# B&R Automation Studio project AAU12Segmenter (part 8)

#### mxA_Start.st
```iecst
ACTION mxA_Start:

	/////////////////////////////////////////////////////
	// Logic to call the KRC_Initialize				   //
	// KRC_Initialize gives back the Status of the	   //
	// like, online, Initialized,.......			   //
	/////////////////////////////////////////////////////

	KRC_Initialize_0.AxisGroupIdx 			:= 1;
	KRC_Initialize_0.KRC_AxisGroupRefArr 	:= ADR(AxisRef);
	HMI_R1_Init_Done 						:=	KRC_Initialize_0.Done;
	HMI_R1_Init_Error 						:=	KRC_Initialize_0.Error;
	HMI_R1_Init_Error_ID 					:=	KRC_Initialize_0.ErrorID;

	KRC_Initialize_0();

	KRC_Initialize_1.AxisGroupIdx 			:= 2;
	KRC_Initialize_1.KRC_AxisGroupRefArr 	:= ADR(AxisRef);
	HMI_R2_Init_Done 						:=	KRC_Initialize_1.Done;
	HMI_R2_Init_Error 						:=	KRC_Initialize_1.Error;
	HMI_R2_Init_Error_ID 					:=	KRC_Initialize_1.ErrorID;

	KRC_Initialize_1();

	/////////////////////////////////////////////////////
	// Logic to call the KRC_Error     			       //
	// KRC_Error gives back the Status of the Robot    //
	// like, online, Initialized,.......			   //
	/////////////////////////////////////////////////////

	KRC_Error_0.AxisGroupIdx 				:= 1;
	KRC_Error_0.MessageReset 				:= HMI_R1_MessageReset;
	KRC_Error_0.KRC_AxisGroupRefArr			:= ADR(AxisRef);
	HMI_R1_Error_General					:= KRC_Error_0.Error;
	HMI_R1_Error_General_ID					:= KRC_Error_0.ErrorID;
	HMI_R1_Error_Activ						:= KRC_Error_0.KrcErrorActive;
	HMI_R1_Error_DrivesNotReady				:= KRC_Error_0.DrivesNotReady;

	KRC_Error_0();

	KRC_Error_1.AxisGroupIdx 				:= 2;
	KRC_Error_1.MessageReset 				:= HMI_R2_MessageReset;
	KRC_Error_1.KRC_AxisGroupRefArr			:= ADR(AxisRef);
	HMI_R2_Error_General					:= KRC_Error_1.Error;
	HMI_R2_Error_General_ID					:= KRC_Error_1.ErrorID;
	HMI_R2_Error_Activ						:= KRC_Error_1.KrcErrorActive;
	HMI_R2_Error_DrivesNotReady				:= KRC_Error_1.DrivesNotReady;

	KRC_Error_1();

	//////////////////////////////////////////////////////
	// KRC_AutomaticExternal allows to control the 		//
	// Robot with the PLC								//
	//////////////////////////////////////////////////////

	KRC_AutomaticExternal_0.AxisGroupIdx 		:= 1;
	KRC_AutomaticExternal_0.MOVE_ENABLE 		:= TRUE;
	KRC_AutomaticExternal_0.DRIVES_OFF 			:= TRUE;
	KRC_AutomaticExternal_0.KRC_AxisGroupRefArr	:= ADR(AxisRef);
	KRC_AutomaticExternal_0.EXT_START 			:= HMI_R1_EXT_START;
	KRC_AutomaticExternal_0.ENABLE_T1 			:= TRUE;
	KRC_AutomaticExternal_0.ENABLE_EXT 			:= TRUE;

	KRC_AutomaticExternal_0();

	KRC_AutomaticExternal_1.AxisGroupIdx 		:= 2;
	KRC_AutomaticExternal_1.MOVE_ENABLE 		:= TRUE;
	KRC_AutomaticExternal_1.DRIVES_OFF 			:= TRUE;
	KRC_AutomaticExternal_1.KRC_AxisGroupRefArr := ADR(AxisRef);
	KRC_AutomaticExternal_1.EXT_START			:= HMI_R2_EXT_START;
	KRC_AutomaticExternal_1.ENABLE_T1 			:= TRUE;
	KRC_AutomaticExternal_1.ENABLE_EXT 			:= TRUE;

	KRC_AutomaticExternal_1();

	//////////////////////////////////////////////////////
	//Function Block for StartUp of Robot				//
	//////////////////////////////////////////////////////

	KRC_AutoStart_0.AxisGroupIdx 				:= 1;
	KRC_AutoStart_0.KRC_AxisGroupRefArr 		:= ADR(AxisRef);
	KRC_AutoStart_0.ExecuteReset 				:= HMI_R1_AutoStart ;

	KRC_AutoStart_0();

	KRC_AutoStart_1.AxisGroupIdx 				:= 2;
	KRC_AutoStart_1.KRC_AxisGroupRefArr 		:= ADR(AxisRef);
	KRC_AutoStart_1.ExecuteReset 				:= HMI_R2_AutoStart ;

	KRC_AutoStart_1();

	//////////////////////////////////////////////////////
	// KRC_SetOverride used to set the Override 		//
	// for the Robot Velocity							//
	//////////////////////////////////////////////////////

	KRC_SetOverride_0.AxisGroupIdx 				:= 1;
	KRC_SetOverride_0.KRC_AxisGroupRefArr 		:= ADR(AxisRef);
	KRC_SetOverride_0.Override 					:= HMI_R1_Override;

	KRC_SetOverride_0();

	KRC_SetOverride_1.AxisGroupIdx 				:= 2;
	KRC_SetOverride_1.KRC_AxisGroupRefArr 		:= ADR(AxisRef);
	KRC_SetOverride_1.Override 					:=HMI_R2_Override;

	KRC_SetOverride_1();

	//////////////////////////////////////////////////////
	//KRC_Diag gives back some information about the 	//
	//axis and robot									//
	//////////////////////////////////////////////////////

	KRC_Diag_0.AxisGroupIdx 					:= 1;
	KRC_Diag_0.KRC_AxisGroupRefArr 				:= ADR(AxisRef);
	KRC_Diag_0.ShowTrace 						:= FALSE;

	KRC_Diag_0();

	KRC_Diag_1.AxisGroupIdx 					:= 2;
	KRC_Diag_1.KRC_AxisGroupRefArr 				:= ADR(AxisRef);
	KRC_Diag_1.ShowTrace 						:= FALSE;

	KRC_Diag_1();

	//////////////////////////////////////////////////////
	//Checking status of KRC and PLC for creating the   //
	//signals for the HMI 								//
	//										 			//
	//////////////////////////////////////////////////////

	CASE HMI_AxisGroup OF

	//////////////////////////////////////////////////////
	//ROBOT 1											//
	//////////////////////////////////////////////////////

		1:
			IF KRC_Diag_0.ProconosCyc_Act = -1 OR KRC_Error_0.NoHeartbeatPCOS THEN
				Status_P := FALSE;
			ELSE
				Status_P := TRUE;
			END_IF

			IF KRC_Diag_0.SubmitCyc_Act = -1 OR KRC_Error_0.NoHeartbeatKRC THEN
				Status_S := FALSE;
			ELSE
				Status_S := TRUE;
			END_IF

			IF KRC_AutomaticExternal_0.EXT THEN
				Status_EXT := 1;
			ELSE
				Status_EXT := 0;
			END_IF

			IF NOT KRC_Error_0.DrivesNotReady AND KRC_AutomaticExternal_0.RC_RDY1 THEN
				Status_I := 1;
			ELSE
				Status_I := 0;
			END_IF

			IF KRC_AutoStart_0.DispActive THEN
				Status_R	:= 1;
			ELSE
				Status_R	:= 0;
			END_IF

	//////////////////////////////////////////////////////
	//ROBOT 2											//
	//////////////////////////////////////////////////////

		2:
			IF KRC_Diag_1.ProconosCyc_Act = -1 OR KRC_Error_1.NoHeartbeatPCOS THEN
				Status_P := FALSE;
			ELSE
				Status_P := TRUE;
			END_IF

			IF KRC_Diag_1.SubmitCyc_Act = -1 OR KRC_Error_1.NoHeartbeatKRC THEN
				Status_S := FALSE;
			ELSE
				Status_S := TRUE;
			END_IF

			IF KRC_AutomaticExternal_1.EXT THEN
				Status_EXT := 1;
			ELSE
				Status_EXT := 0;
			END_IF

			IF NOT KRC_Error_1.DrivesNotReady AND KRC_AutomaticExternal_1.RC_RDY1 THEN
				Status_I := 1;
			ELSE
				Status_I := 0;
			END_IF

			IF KRC_AutoStart_1.DispActive THEN
				Status_R	:= 1;
			ELSE
				Status_R	:= 0;
			END_IF

	//////////////////////////////////////////////////////
	//ROBOT 3,4,5										//
	//////////////////////////////////////////////////////

		3,4,5:

			Status_P := FALSE;
			Status_S := FALSE;
			Status_I := 0;
			Status_R := 0;
			Status_EXT := 0;

	END_CASE;

END_ACTION
```

#### mxA_LinearMovement.st
```iecst
ACTION mxA_LinearMovement:

	CASE pState OF

		0:
			// Waiting for robot 1 to be ready to move
			IF 	Status_P > 0 AND Status_S > 0 AND Status_I > 0 AND Status_R > 0 AND Status_EXT > 0 THEN
				pState := 20;
			END_IF

		10:
			toolCover.X := 0;
			toolCover.Y := 0;
			toolCover.Z := 100;
			toolCover.A := 0;
			toolCover.B := 0;
			toolCover.C := 0;

			KRC_WriteToolData_0.AxisGroupIdx 		:= HMI_AxisGroup;
			KRC_WriteToolData_0.KRC_AxisGroupRefArr := ADR(AxisRef);
			KRC_WriteToolData_0.ToolNo 				:= 1;
			KRC_WriteToolData_0.ToolData 			:= toolCover;
			KRC_WriteToolData_0.BufferMode 			:= 2;
			KRC_WriteToolData_0.ExecuteCmd			:= TRUE;

			IF KRC_WriteToolData_0.Done THEN
				KRC_WriteToolData_0.ExecuteCmd		:= FALSE;
				pState := 20;
			END_IF

		20:

			//Set frames as coordsys
			mxa_ValuesToCOORDSYS_0.Tool 	:= 1; // Change to 1 when it works
			mxa_ValuesToCOORDSYS_0.Base 	:= 1;
			mxa_ValuesToCOORDSYS_0.IPO_Mode := 0;

			pState := 30;

		30:

			coordSys := mxa_ValuesToCOORDSYS_0.COORDSYS;

			KRC_MoveLinearAbsolute_0.AxisGroupIdx 			:= HMI_AxisGroup;
			KRC_MoveLinearAbsolute_0.KRC_AxisGroupRefArr	:= ADR(AxisRef);
			KRC_MoveLinearAbsolute_0.Velocity				:= 10;
			KRC_MoveLinearAbsolute_0.Acceleration  			:= 20;
			KRC_MoveLinearAbsolute_0.CoordinateSystem		:= coordSys;
			KRC_MoveLinearAbsolute_0.OriType 				:= 0;
			KRC_MoveLinearAbsolute_0.BufferMode				:= 2;

			pState := 40;

		40:
			endPOS.X := 302;
			endPOS.Y := -2;
			endPOS.Z := 527;
			endPOS.A := -178;
			endPOS.B := 26;
			endPOS.C := -178;
			endPOS.Status := 2; //010
			endPOS.Turn := 2; //000010

			KRC_MoveLinearAbsolute_0.Position			:= endPOS;

			KRC_MoveLinearAbsolute_0.ExecuteCmd 		:= TRUE;
			IF KRC_MoveLinearAbsolute_0.Done THEN
				KRC_MoveLinearAbsolute_0.ExecuteCmd 	:= FALSE;
				pState 									:= 50;
			END_IF

		50:
			endPOS.X := 430;
			endPOS.Y := -2;
			endPOS.Z := 527;
			endPOS.A := -178;
			endPOS.B := 26;
			endPOS.C := -178;
			endPOS.Status := 2; //010
			endPOS.Turn := 2; //000010

			KRC_MoveLinearAbsolute_0.Position			:= endPOS;

			KRC_MoveLinearAbsolute_0.ExecuteCmd 		:= TRUE;
			IF KRC_MoveLinearAbsolute_0.Done THEN
				KRC_MoveLinearAbsolute_0.ExecuteCmd 	:= FALSE;
				pState 									:= 40;
			END_IF

	END_CASE

	KRC_WriteToolData_0();
	mxa_ValuesToCOORDSYS_0();
	KRC_MoveLinearAbsolute_0();

END_ACTION
```

### Variables.var - Global variables
```iecst
(*********************************************************************************
 * Copyright: Bernecker + Rainer
 * Author:    reschl
 * Created:   July 02, 2015/4:23 PM
 *********************************************************************************
 * Global variables of project
 *********************************************************************************)
(*KRC <----> PLC communication*)
VAR
	KRC_Input : ARRAY[0..5,0..253] OF BYTE;
	KRC_Output : ARRAY[0..5,0..253] OF BYTE;
	InputVariables : ARRAY[0..5,0..253] OF USINT;
	OutputVariables : ARRAY[0..5,0..253] OF USINT;
	KUKAs : ARRAY[0..5] OF KUKA;
	KRC4_Input_1 : ARRAY[0..254] OF BYTE; (*Variable with the BYTE information from KRC*)
	KRC4_Input : ARRAY[0..254] OF BYTE; (*Variable with the BYTE information from KRC*)
	KRC4_Output_1 : ARRAY[0..254] OF BYTE; (*Variable with the BYTE information to KRC*)
	KRC4_Output : ARRAY[0..254] OF BYTE; (*Variable with the BYTE infromation to KRC*)
	InputVariablePL_1 : ARRAY[0..255] OF USINT;
	InputVariablePL : ARRAY[0..255] OF USINT;
	OutputVariablePL_1 : ARRAY[0..255] OF USINT;
	OutputVariablePL : ARRAY[0..255] OF USINT;
END_VAR
(*PositonArray, Coordsys etc*)
VAR RETAIN
	TeachPosition : POSITION_ARRAY; (*TeachingPositions -> retain to be save when restarting*)
END_VAR
VAR
	JogPosAxis : E6AXIS := (A2:=-90,A3:=90);
	JoggingCoordSys : COORDSYS; (*Variable for the CoordSystem when Jogging*)
	Coordsys_1 : COORDSYS;
END_VAR
VAR RETAIN
	gParameter : USINT;
END_VAR
(*HMI Variablen*)
VAR
	gCurrentPage : INT; (*Shows current page index of the Visualization*)
	HMI_Base_act : INT;
	HMI_Tool_act : INT;
	HMI_ExeAbort : BOOL;
	HMI_ExeMoveDirect : BOOL;
	HMI_AxisGroup : INT;
	HMI_R2_MessageReset : BOOL;
	HMI_R2_Override : INT;
	HMI_R2_AutoStart : BOOL;
	HMI_R2_EXT_START : BOOL;
	HMI_R2_Error_DrivesNotReady : BOOL;
	HMI_R2_Error_Activ : BOOL;
	HMI_R2_Error_General_ID : DINT;
	HMI_R2_Error_General : BOOL;
	HMI_R2_Init_Error_ID : DINT;
	HMI_R2_Init_Error : BOOL;
	HMI_R2_Init_Done : BOOL;
	HMI_R1_MessageReset : BOOL;
	HMI_R1_Override : INT;
	HMI_R1_AutoStart : BOOL;
	HMI_R1_EXT_START : BOOL;
	HMI_R1_Error_DrivesNotReady : BOOL;
	HMI_R1_Error_Activ : BOOL;
	HMI_R1_Error_General_ID : DINT;
	HMI_R1_Error_General : BOOL;
	HMI_R1_Init_Error_ID : DINT;
	HMI_R1_Init_Error : BOOL;
	HMI_R1_Init_Done : BOOL;
	HMI_A6 : REAL;
	HMI_A5 : REAL;
	HMI_A4 : REAL;
	HMI_A3 : REAL;
	HMI_A2 : REAL;
	HMI_A1 : REAL;
	HMI_C : REAL;
	HMI_B : REAL;
	HMI_A : REAL;
	HMI_Z : REAL;
	HMI_Y : REAL;
	HMI_X : REAL;
	HMI_A6_C_M : BOOL;
	HMI_A6_C_P : BOOL;
	HMI_A5_B_M : BOOL;
	HMI_A5_B_P : BOOL;
	HMI_A4_A_M : BOOL;
	HMI_A4_A_P : BOOL;
	HMI_A3_Z_M : BOOL;
	HMI_A3_Z_P : BOOL;
	HMI_A2_Y_M : BOOL;
	HMI_A2_Y_P : BOOL;
	HMI_A1_X_M : BOOL;
	HMI_A1_X_P : BOOL;
	HMI_Increment : INT;
	HMI_MoveType : INT;
END_VAR
```

### Types.typ - Global data types
```iecst
TYPE
	KUKA : 	STRUCT
		cm : brdkCM; (*Change type after integration into Smart Lab project*)
		init : init_function;
		motion : motion_function;
		read : read_function;
		operationType : operation_type;
		gripperType : gripper_type;
		TON_Timer : TON;
		operationDone : BOOL := FALSE; (*Maybe don't need. Depends how we send finish flag to ACOPOS*)
		status : status;
	END_STRUCT;
	init_function : 	STRUCT
		KRC_ReadAxisGroup : KRC_ReadAxisGroup;
		KRC_Initialize : KRC_Initialize;
		KRC_Error : KRC_Error;
		KRC_AutomaticExternal : KRC_AutomaticExternal;
		KRC_AutoStart : KRC_AutoStart;
		KRC_SetOverride : KRC_SetOverride;
		KRC_Diag : KRC_Diag;
		KRC_WriteAxisGroup : KRC_WriteAxisGroup;
	END_STRUCT;
	motion_function : 	STRUCT
		KRC_MoveDirectAbsolute : KRC_MoveDirectAbsolute;
		KRC_MoveDirectRelative : KRC_MoveDirectRelative;
		KRC_MoveLinearAbsolute : KRC_MoveLinearAbsolute;
		KRC_MoveLinearRelative : KRC_MoveLinearRelative;
	END_STRUCT;
	read_function : 	STRUCT
		KRC_ReadActualPosition : KRC_ReadActualPosition;
		KRC_ReadActualAxisPosition : KRC_ReadActualAxisPosition;
	END_STRUCT;
	operation_type :
		(
		ASSEMBLY := 0,
		PROCESS := 1
		);
	gripper_type :
		(
		COVER_GRIPPER := 0,
		PCB_GRIPPER := 1,
		FUSE_GRIPPER := 2
		);
	status : 	STRUCT
		S_ : BOOL;
		I_ : BOOL;
		R_ : BOOL;
		EXT_ : BOOL;
		P_ : BOOL;
	END_STRUCT;
END_TYPE
```

### Program Logical/Modules/KUKA/KUKA (IEC)

#### Types.typ - Local data types
```iecst
TYPE
	KUKA : 	STRUCT
		axisGroupIdx : USINT;
		startState : USINT;
		cm : brdkCM;
		start : start_function;
		motion : motion_function;
		convert : convert_function;
		read : read_function;
		write : write_function;
		status : status;
		operationType : operation_type;
		eeType : end_effector_type;
		gripperAction : GripperAction;
		tempPosition : E6POS;
		TON : TON;
	END_STRUCT;
	start_function : 	STRUCT
		KRC_Initialize : KRC_Initialize;
		KRC_Error : KRC_Error;
		KRC_AutomaticExternal : KRC_AutomaticExternal;
		KRC_AutoStart : KRC_AutoStart;
		KRC_SetOverride : KRC_SetOverride;
		KRC_Diag : KRC_Diag;
		KRC_Abort : KRC_Abort;
	END_STRUCT;
	motion_function : 	STRUCT
		KRC_MoveDirectAbsolute : KRC_MoveDirectAbsolute; (*PTP absolute motion*)
		KRC_MoveDirectRelative : KRC_MoveDirectRelative; (*PTP relative motion*)
		KRC_MoveLinearAbsolute : KRC_MoveLinearAbsolute; (*LIN absolute motion*)
		KRC_MoveLinearRelative : KRC_MoveLinearRelative; (*LIN relative motion*)
		KRC_MoveAxisAbsolute : KRC_MoveAxisAbsolute; (*JOINT absolute motion*)
	END_STRUCT;
	convert_function : 	STRUCT
		ValuesToCOORDSYS : mxa_ValuesToCOORDSYS;
		ValuesToPosition : ValuesToPosition;
		ValuesToMagazineFrame : ValuesToMagazineFrame;
	END_STRUCT;
	read_function : 	STRUCT
		KRC_ReadAxisGroup : KRC_ReadAxisGroup;
		KRC_ReadActualPosition : KRC_ReadActualPosition;
		KRC_ReadActualAxisPosition : KRC_ReadActualAxisPosition;
	END_STRUCT;
	write_function : 	STRUCT
		KRC_WriteAxisGroup : KRC_WriteAxisGroup;
		KRC_WriteToolData : KRC_WriteToolData;
		KRC_WriteBaseData : KRC_WriteBaseData;
	END_STRUCT;
	status : 	STRUCT
		S_ : BOOL;
		I_ : BOOL;
		R_ : BOOL;
		EXT_ : BOOL;
		P_ : BOOL;
	END_STRUCT;
	operation_type :
		(
		ASSEMBLY := 0,
		PROCESS := 1
		);
	end_effector_type :
		(
		COVER_EE := 1,
		PCB_EE := 2,
		FUSE_EE := 3,
		DRILL_EE := 4
		);
	gripper_action_type :
		(
		OPEN := 0,
		CLOSE := 1
		);
	robot_position_type :
		(
		DEFAULT := 0,
		APPROACH_MAGAZINE := 1,
		APPROACH_WORKSTATION := 2
		);
END_TYPE
```

#### Variables.var - Local variables
```iecst
VAR
	KUKAs : ARRAY[0..5] OF KUKA;
END_VAR
(*AxisStructure*)
VAR
	AxisRef : AXIS_GROUP_REF_ARR; (*Axis Reference of the Robot*)
END_VAR
(*Instance of FB*)
VAR
	mxa_ValuesToCOORDSYS_0 : mxa_ValuesToCOORDSYS;
	EETypeToFrame_0 : EETypeToFrame;
END_VAR
(*Variables for UDP-communication*)
VAR
	i : USINT; (*IndexVariable for ErrorMessages*)
	InputUDPString : STRING[255]; (*Variable with Message from KRC*)
	counterMsg : INT;
	WorkAroundCounter : INT;
	step_UDPConnect : INT; (*State-Variable for Errorhandling*)
	TextArray : ARRAY[0..15] OF STRING[255]; (*TextArray contains Messages from KRC*)
	UdpOpen_0 : UdpOpen; (*FunctionBlock to Open Port*)
	UdpOpen_1 : UdpOpen; (*FunctionBlock to Open Port*)
	UdpRecv_0 : UdpRecv; (*FunctionBlock to Receive Message*)
	UdpSend_0 : UdpSend; (*FunctionBlock to Send Message*)
	MsgToKrc : STRING[17]; (*Contains the Message which is send to KRC for getting all Messages*)
	ReloadMsg : BOOL; (*Variable triggers the Sequence to get Messages*)
END_VAR
VAR CONSTANT
	STATE_DISPLAY : INT := 5; (*STATE to display the Message*)
	STATE_RECEIVE : INT := 3; (*STATE to receive a new Message*)
	STATE_OPEN : INT := 0; (*STATE for opening the Ports*)
	STATE_SEND : INT := 2; (*STATE for sending a request to KRC*)
	STATE_WAIT : INT := 1; (*STATE for Waiting to trigger a new Request*)
END_VAR
VAR
	TON_0 : TON;
END_VAR
(*Misc*)
VAR
	acoposBase : FRAME;
	bottomCoverMagazineBase : FRAME;
	pcbMagazineBase : FRAME;
	fuseMagazineBase : FRAME;
	topCoverMagazineBase : FRAME;
	unloadingBase : FRAME;
	coordSys : COORDSYS;
	endPOS : E6POS;
	position1 : E6AXIS;
	position2 : E6AXIS;
END_VAR
(*For robot operations*)
VAR
	gripperWaitTime : INT;
END_VAR
VAR CONSTANT
	relativeDistance : REAL := 80.0;
	relativeDrillDistance : REAL := 10.0;
END_VAR
VAR
	drillYOffset : REAL := 27*2;
	drillXOffset : REAL := 53*2;
	numDoneHoles : USINT := 0;
	fusePickOffset : REAL := 13; (*Distance between fuses*)
	k : INT;
END_VAR
VAR CONSTANT
	unloadSizeX : INT := 2;
	unloadSizeY : INT := 2;
	unloadSizeZ : INT := 4;
END_VAR
VAR
	stackCounter : ARRAY[0..1,0..1] OF INT := [4(0)];
	idAtStack : ARRAY[0..1,0..1] OF INT := [4(-1)];
	xIdx : INT;
	yIdx : INT;
	xIdxTemp : INT := -1;
	yIdxTemp : INT := -1;
	orderCounter : ARRAY[0..1,0..1] OF INT := [4(0)];
END_VAR
(*References*)
VAR
	pKuka : REFERENCE TO KUKA;
	cm : REFERENCE TO brdkCM;
END_VAR
(*Variable mapping*)
VAR
	orderAmount : SINT;
	orderSpec : ARRAY[0..5] OF SINT;
	robotExecute : ARRAY[0..5] OF BOOL;
	robotDone : ARRAY[0..5] OF BOOL;
	robotBusy : ARRAY[0..5] OF BOOL;
END_VAR
```

#### Main.st - Cyclic code
```iecst
PROGRAM _INIT

	FOR i := 0 TO 5 DO
		KUKAs[i].axisGroupIdx := i + 1;
		KUKAs[i].gripperAction.whitePin := ADR(gripperWhitePins[i]);
		KUKAs[i].gripperAction.blackPin := ADR(gripperBlackPins[i]);
		KUKAs[i].gripperAction.action := OPEN;
		KUKAs[i].gripperAction();
		KUKAs[i].cm.state := 0;
		KUKAs[i].startState := 0;
	END_FOR

	// Setting end-effector type
	KUKAs[0].eeType := COVER_EE;
	KUKAs[1].eeType := DRILL_EE;
	KUKAs[2].eeType := PCB_EE;
	KUKAs[3].eeType := FUSE_EE;
	KUKAs[4].eeType := COVER_EE;
	KUKAs[5].eeType := COVER_EE;

	// Setting the operation type
	KUKAs[0].operationType := ASSEMBLY;
	KUKAs[1].operationType := PROCESS;
	KUKAs[2].operationType := ASSEMBLY;
	KUKAs[3].operationType := ASSEMBLY;
	KUKAs[4].operationType := ASSEMBLY;
	KUKAs[5].operationType := HANDLING;

	gripperWaitTime := 250; // in ms

END_PROGRAM

PROGRAM _CYCLIC

	FOR i := 0 TO 5 DO // CHANGE TO 0 TO 5 WHEN ALL ROBOTS WORK

		// Accessing the specific KUKA for easier naming
		pKuka ACCESS ADR(KUKAs[i]);
		cm ACCESS ADR(KUKAs[i].cm);

		// Logic to transform USINT (Input) to BYTE (FUBS)
		brsmemcpy(ADR(KRC_Input[0]), ADR(InputVariables[i,0]), 254);

		/////////////////////////////////////////////////////
		// KRC_ReadAxisGroup has to be called at the Begin //
		// of the Cyclic Task to get all the Information   //
		// From the KRC from all KUKAs					   //
		/////////////////////////////////////////////////////

		pKuka.read.KRC_ReadAxisGroup.KRC4_Input 			:= ADR(KRC_Input);
		pKuka.read.KRC_ReadAxisGroup.AxisGroupIdx 			:= pKuka.axisGroupIdx;
		pKuka.read.KRC_ReadAxisGroup.KRC_AxisGroupRefArr 	:= ADR(AxisRef);

		pKuka.read.KRC_ReadAxisGroup();

		// RobotStart contains FB calls associated with initialization of the robots and diagnosis
		RobotStart;

		//robotDone[0] := robotDone[1] := robotDone[2] := robotDone[3] := robotDone[4] := robotDone[5] := TRUE; // ALSO CHANGE IN ROBOTEXECUTE IN ACOPOS!!!
		robotDone[5] := TRUE;

		// If the robot is ready, begin actual program
		IF 	pKuka.status.P_ AND pKuka.status.S_ AND pKuka.status.R_ AND pKuka.status.I_ AND pKuka.status.EXT_ THEN
			CASE cm.state OF
				0: // INITIALIZING
					pKuka.convert.ValuesToCOORDSYS.Tool := 1;
					pKuka.convert.ValuesToPosition.axisGroupIdx := pKuka.axisGroupIdx;

					pKuka.motion.KRC_MoveDirectAbsolute.AxisGroupIdx := pKuka.motion.KRC_MoveLinearAbsolute.AxisGroupIdx := pKuka.motion.KRC_MoveLinearRelative.AxisGroupIdx
						:=  pKuka.axisGroupIdx;
					pKuka.motion.KRC_MoveDirectAbsolute.KRC_AxisGroupRefArr := pKuka.motion.KRC_MoveLinearAbsolute.KRC_AxisGroupRefArr := pKuka.motion.KRC_MoveLinearRelative.KRC_AxisGroupRefArr
					:= ADR(AxisRef);

					pKuka.motion.KRC_MoveDirectAbsolute.Velocity := pKuka.motion.KRC_MoveLinearAbsolute.Velocity := pKuka.motion.KRC_MoveLinearRelative.Velocity
						:= 100; // Velocity in percent

					pKuka.motion.KRC_MoveDirectAbsolute.Acceleration := pKuka.motion.KRC_MoveLinearAbsolute.Acceleration := pKuka.motion.KRC_MoveLinearRelative.Acceleration
						:= 50; // Acceleration in percent
					pKuka.motion.KRC_MoveDirectAbsolute.BufferMode := pKuka.motion.KRC_MoveLinearAbsolute.BufferMode := pKuka.motion.KRC_MoveLinearRelative.BufferMode
						:= 2; // BUFFERED
					pKuka.motion.KRC_MoveLinearAbsolute.OriType := pKuka.motion.KRC_MoveLinearRelative.OriType
						:= 0; // 0: VAR | 1: CONSTANT | 2: JOINT
					pKuka.motion.KRC_MoveDirectAbsolute.ExecuteCmd := pKuka.motion.KRC_MoveLinearAbsolute.ExecuteCmd := pKuka.motion.KRC_MoveLinearRelative.ExecuteCmd
						:= FALSE;

					cm.state := 101;

				100..499: // SETTING TOOL AND BASE DATA
					WriteToolData; // 101..200
					WriteBaseData; // 201..300

				500..999: // Move robot to home position (position depends on operation type)
					RobotHoming;

				1000..1999: // RUNNING MANIPULATOR PROGRAMS

					CASE pKuka.operationType OF
						ASSEMBLY:
							RobotAssembly;

						PROCESS:
							RobotProcess;

						HANDLING:
							RobotHandling;
					END_CASE
			END_CASE

		END_IF

		//Calling function blocks to update content
		pKuka.motion.KRC_MoveLinearAbsolute();
		pKuka.motion.KRC_MoveLinearRelative();
		pKuka.motion.KRC_MoveDirectAbsolute();
		pKuka.gripperAction();
		pKuka.TON();

		/////////////////////////////////////////////////////
		// FunctionBlock to write the Output on the Struct //
		/////////////////////////////////////////////////////

		pKuka.write.KRC_WriteAxisGroup.AxisGroupIdx			:= pKuka.axisGroupIdx;
		pKuka.write.KRC_WriteAxisGroup.KRC_AxisGroupRefArr 	:= ADR(AxisRef);
		pKuka.write.KRC_WriteAxisGroup.KRC4_Output 			:= ADR(KRC_Output);

		pKuka.write.KRC_WriteAxisGroup();

		// Logic to transform BYTE (FUBS) to USINT (Input)
		brsmemcpy(ADR(OutputVariables[i,0]), ADR(KRC_Output[0]), 254);

	END_FOR

END_PROGRAM
```

#### RobotStart.st
```iecst
ACTION RobotStart:

	CASE pKuka.startState OF

		0: // Configuring KUKA FBs once

			// Logic to call the KRC_Initialize
			pKuka.start.KRC_Initialize.AxisGroupIdx 				:= pKuka.axisGroupIdx;
			pKuka.start.KRC_Initialize.KRC_AxisGroupRefArr 			:= ADR(AxisRef);

			// Logic to call the KRC_Error
			pKuka.start.KRC_Error.AxisGroupIdx 						:= pKuka.axisGroupIdx;
			pKuka.start.KRC_Error.MessageReset 						:= FALSE; // REMEMBER TO CHANGE LATER
			pKuka.start.KRC_Error.KRC_AxisGroupRefArr				:= ADR(AxisRef);

			// Logic to call KRC_AutomaticExternal
			pKuka.start.KRC_AutomaticExternal.AxisGroupIdx 			:= pKuka.axisGroupIdx;
			pKuka.start.KRC_AutomaticExternal.MOVE_ENABLE 			:= TRUE;
			pKuka.start.KRC_AutomaticExternal.DRIVES_OFF 			:= TRUE;
			pKuka.start.KRC_AutomaticExternal.KRC_AxisGroupRefArr	:= ADR(AxisRef);
			pKuka.start.KRC_AutomaticExternal.EXT_START 			:= FALSE; // Binded to Continue Prog in original program
			pKuka.start.KRC_AutomaticExternal.ENABLE_T1 			:= TRUE;
			pKuka.start.KRC_AutomaticExternal.ENABLE_EXT 			:= TRUE;

			// Logic for startup of robot
			pKuka.start.KRC_AutoStart.AxisGroupIdx 					:= pKuka.axisGroupIdx;
			pKuka.start.KRC_AutoStart.KRC_AxisGroupRefArr 			:= ADR(AxisRef);
			pKuka.start.KRC_AutoStart.ExecuteReset 					:= FALSE; // REMEMBER TO CHANGE LATER

			// Logic to set override for robot velocity
			pKuka.start.KRC_SetOverride.AxisGroupIdx 				:= pKuka.axisGroupIdx;
			pKuka.start.KRC_SetOverride.KRC_AxisGroupRefArr 		:= ADR(AxisRef);
			pKuka.start.KRC_SetOverride.Override 					:= 10; // REMEMBER TO CHANGE LATER

			// Logic to set
			pKuka.start.KRC_Abort.AxisGroupIdx 						:= pKuka.axisGroupIdx;
			pKuka.start.KRC_Abort.KRC_AxisGroupRefArr				:= ADR(AxisRef);
			pKuka.start.KRC_Abort.ExecuteCmd						:= FALSE;  /// Used to be set by HMI - Remember to incorporate it later

			// Logic to set KRC_Diag
			pKuka.start.KRC_Diag.AxisGroupIdx 						:= pKuka.axisGroupIdx;
			pKuka.start.KRC_Diag.KRC_AxisGroupRefArr 				:= ADR(AxisRef);
			pKuka.start.KRC_Diag.ShowTrace 							:= FALSE;

			pKuka.startState := 1;

		1: // Wait for P, S and EXT
			IF pKuka.status.P_ AND pKuka.status.S_ AND pKuka.status.EXT_ THEN
				pKuka.startState := 2;
			END_IF

		2: // Reset KRC errors and autostart
			pKuka.start.KRC_Error.MessageReset := TRUE;
			pKuka.start.KRC_AutoStart.ExecuteReset := TRUE;

			IF pKuka.status.R_ AND pKuka.status.I_ THEN
				pKuka.start.KRC_Error.MessageReset := FALSE;
				pKuka.start.KRC_AutoStart.ExecuteReset := FALSE;
				pKuka.startState := 3;
			END_IF

		3: // Check if any error occurred
			IF 	NOT pKuka.status.P_ OR
				NOT pKuka.status.S_ OR
				NOT pKuka.status.EXT_ OR
				NOT pKuka.status.R_ OR
				NOT pKuka.status.I_ THEN

				pKuka.startState := 1;

			END_IF

	END_CASE

	// Logic to call the KRC_Initialize
	// KRC_Initialize gives back the Status OF the like, online, Initialized,.......
	pKuka.start.KRC_Initialize();

	// Logic to call the KRC_Error.
	// KRC_Error gives back the Status OF the Robot like, online, Initialized,.......
	pKuka.start.KRC_Error();

	// KRC_AutomaticExternal allows to control the Robot with the PLC
	pKuka.start.KRC_AutomaticExternal();

	//Function Block for StartUp of Robot
	pKuka.start.KRC_AutoStart();

	// KRC_SetOverride used to set the Override for the Robot Velocity
	pKuka.start.KRC_SetOverride();

	// KRC_Abort cancels all active and buffered statements and motions
	pKuka.start.KRC_Abort();

	// KRC_Diag gives back some information about the axis and robot
	pKuka.start.KRC_Diag();

	//Checking status of KRC and PLC for creating the signals for the HMI
	IF pKuka.start.KRC_Diag.ProconosCyc_Act = -1 OR pKuka.start.KRC_Error.NoHeartbeatPCOS THEN
		pKuka.status.P_ := FALSE;
	ELSE
		pKuka.status.P_ := TRUE;
	END_IF

	IF pKuka.start.KRC_Diag.SubmitCyc_Act = -1 OR pKuka.start.KRC_Error.NoHeartbeatKRC THEN
		pKuka.status.S_ := FALSE;
	ELSE
		pKuka.status.S_ := TRUE;
	END_IF

	IF pKuka.start.KRC_AutomaticExternal.EXT THEN
		pKuka.status.EXT_ := TRUE;
	ELSE
		pKuka.status.EXT_ := FALSE;
	END_IF

	IF NOT pKuka.start.KRC_Error.DrivesNotReady AND pKuka.start.KRC_AutomaticExternal.RC_RDY1 THEN
		pKuka.status.I_ := TRUE;
	ELSE
		pKuka.status.I_ := FALSE;
	END_IF

	IF pKuka.start.KRC_AutoStart.DispActive THEN
		pKuka.status.R_	:= TRUE;
	ELSE
		pKuka.status.R_	:= FALSE;
	END_IF

END_ACTION
```

#### ErrorMessage.st
```iecst
ACTION ErrorMessage:

	CASE step_UDPConnect OF

		//////////////////////////////////////////////////////////
		//			Opening the 2 Ports to communicate			//
		//	Port 55555 is used for Receiving					//
		//	Port 50055 is used for Sending						//
		//////////////////////////////////////////////////////////
		STATE_OPEN:
			UdpOpen_0.enable := 1; 										//opening port for Receiving
			UdpOpen_0.port := 55555;
			UdpOpen_0();

			UdpOpen_1.enable := 1;  									//opening port for Sending
			UdpOpen_1.port := 50055;
			UdpOpen_1();

			IF UdpOpen_0.status = ERR_OK AND UdpOpen_1.status = ERR_OK THEN		//if both ports are open send request
				step_UDPConnect := STATE_WAIT;
			END_IF

		//////////////////////////////////////////////////////////
		//		Waiting State for the manual trigger			//
		//		to get all the Messages	 (request)				//
		//////////////////////////////////////////////////////////
		STATE_WAIT:

			TON_0.IN := 0;

			IF ReloadMsg = 1 OR WorkAroundCounter = 1 THEN				//Var WorkAroundCounter is just a Workaround to Reload the messages 2 times
				step_UDPConnect := STATE_SEND;							// otherwise messages are displayed when requensting the first time!
			END_IF

			IF WorkAroundCounter >= 2 THEN
				WorkAroundCounter := 0;
			END_IF

		//////////////////////////////////////////////////////////
		//		Sending the Message to the KRC to 				//
		//		get all the Messages							//
		//////////////////////////////////////////////////////////
		STATE_SEND:

			FOR counterMsg := 0 TO 15 DO						//Reseting the Array with the Messages
				TextArray[counterMsg] := '';
			END_FOR

			i := 0;												//Reseting counter for the Message Array
			MsgToKrc := 'GetAllKrcMessages';					//Message to KRC -> to get the Messages from KRC

			UdpSend_0.enable := 1;
			UdpSend_0.ident := UdpOpen_1.ident;
			UdpSend_0.pHost := ADR('192.168.1.2');
			UdpSend_0.port := 50055;
			UdpSend_0.pData := ADR(MsgToKrc);
			UdpSend_0.datalen := SIZEOF(MsgToKrc);
			UdpSend_0();

			IF UdpSend_0.status = ERR_OK THEN					//ERR_OK -> NO ERROR
				WorkAroundCounter := WorkAroundCounter +1;
				step_UDPConnect := STATE_RECEIVE;
			END_IF

		//////////////////////////////////////////////////////////
		//		Receiving the Messages from KRC					//
		//		Per cycle 1 msg will be received				//
		// 		If no message after 1s change to STATE_WAIT		//
		//////////////////////////////////////////////////////////
		STATE_RECEIVE:
			UdpRecv_0.enable := 1;
			UdpRecv_0.ident := UdpOpen_0.ident;
			UdpRecv_0.pData := ADR(InputUDPString);
			UdpRecv_0.datamax := 255;
			UdpRecv_0();

			IF UdpRecv_0.status = ERR_OK THEN					//ERR_OK -> NO ERROR

				InputUDPString 	:= LEFT(InputUDPString, UDINT_TO_INT(UdpRecv_0.recvlen));
				TON_0.IN 		:= 0; // Reset timer - msg received
				step_UDPConnect 		:= STATE_DISPLAY;

			ELSIF (UdpRecv_0.status = udpERR_NO_DATA) THEN

				TON_0.IN := 1; // set timer - no msg available, after 1 sec change state to wait
				TON_0.PT := T#1s;

			END_IF

			// check if timer is set to true
			IF TON_0.Q = 1 THEN

				step_UDPConnect := STATE_WAIT;
			END_IF

		//////////////////////////////////////////////////////////
		//		State to transfer the Message					//
		//		to the Array which is displayed at Visu			//
		//////////////////////////////////////////////////////////
		STATE_DISPLAY:

			TextArray[i] := InputUDPString;								//write current message to array to display
			IF i >= 14 THEN
				i := 0;
			ELSE
				memset(ADR(InputUDPString),0,SIZEOF(InputUDPString));	//Clear / Reset the input of the Variable
				i := i + 1;
				step_UDPConnect := STATE_RECEIVE;						//Go to Receive state, to see if another message available
			END_IF;

	END_CASE;

	//Call of the Timer for the TimeOut when no Message
	TON_0();

END_ACTION
```

#### WriteToolData.st
```iecst
ACTION WriteToolData:

	CASE pKuka.cm.state OF
		101: // ToolNo = 1
			EETypeToFrame_0.eeType := pKuka.eeType;
			EETypeToFrame_0();

			pKuka.write.KRC_WriteToolData.AxisGroupIdx 			:= pKuka.axisGroupIdx;
			pKuka.write.KRC_WriteToolData.KRC_AxisGroupRefArr 	:= ADR(AxisRef);
			pKuka.write.KRC_WriteToolData.ToolNo 				:= 1;
			pKuka.write.KRC_WriteToolData.ToolData 				:= EETypeToFrame_0.frame;
			pKuka.write.KRC_WriteToolData.BufferMode 			:= 2;
			pKuka.write.KRC_WriteToolData.ExecuteCmd			:= TRUE;

			IF pKuka.write.KRC_WriteToolData.Done THEN
				pKuka.write.KRC_WriteToolData.ExecuteCmd		:= FALSE;
				pKuka.cm.state := 201;
			END_IF

	END_CASE

	pKuka.write.KRC_WriteToolData();

END_ACTION
```

#### WriteBaseData.st
```iecst
// For now each robot knows all bases even though it only needs to now the ACOPOS6D base and its own magazine base
ACTION WriteBaseData: // Relative to world (can only be used when each robots world has been changed)

	CASE cm.state OF
		201: // ACOPOS6D base (BaseNo = 1)
			acoposBase.X := 240;
			acoposBase.Y := 240;
			acoposBase.Z := 70;
			acoposBase.A := 0;
			acoposBase.B := 0;
			acoposBase.C := 0;

			pKuka.write.KRC_WriteBaseData.AxisGroupIdx 			:= pKuka.axisGroupIdx;
			pKuka.write.KRC_WriteBaseData.KRC_AxisGroupRefArr 	:= ADR(AxisRef);
			pKuka.write.KRC_WriteBaseData.BaseNo 				:= 1;
			pKuka.write.KRC_WriteBaseData.BaseData 				:= acoposBase;
			pKuka.write.KRC_WriteBaseData.BufferMode 			:= 2;
			pKuka.write.KRC_WriteBaseData.ExecuteCmd			:= TRUE;

			IF pKuka.write.KRC_WriteBaseData.Done THEN
				pKuka.write.KRC_WriteBaseData.ExecuteCmd		:= FALSE;

				IF pKuka.operationType = ASSEMBLY THEN
					cm.state := 202;
				ELSIF pKuka.operationType = PROCESS THEN
					cm.state := 500;
				END_IF
			END_IF

		202: // Magazine base (BaseNo = 2)
			pKuka.convert.ValuesToMagazineFrame.axisGroupIdx 	:= pKuka.axisGroupIdx;
			pKuka.convert.ValuesToMagazineFrame();

			pKuka.write.KRC_WriteBaseData.AxisGroupIdx 			:= pKuka.axisGroupIdx;
			pKuka.write.KRC_WriteBaseData.KRC_AxisGroupRefArr 	:= ADR(AxisRef);
			pKuka.write.KRC_WriteBaseData.BaseNo 				:= 2;
			pKuka.write.KRC_WriteBaseData.BaseData 				:= pKuka.convert.ValuesToMagazineFrame.outputFrame;
			pKuka.write.KRC_WriteBaseData.BufferMode 			:= 2;
			pKuka.write.KRC_WriteBaseData.ExecuteCmd			:= TRUE;

			IF pKuka.write.KRC_WriteBaseData.Done THEN
				pKuka.write.KRC_WriteBaseData.ExecuteCmd		:= FALSE;
				cm.state := 500;
			END_IF

	END_CASE

	pKuka.write.KRC_WriteBaseData();

END_ACTION
```

#### RobotHoming.st
```iecst
ACTION RobotHoming:

	// Check if current iteration is drilling manipulator
	CASE pKuka.operationType OF
		ASSEMBLY:
			pKuka.convert.ValuesToPosition.posType := APPROACH_MAGAZINE;

		PROCESS, HANDLING:
			pKuka.convert.ValuesToPosition.posType := APPROACH_WORKSTATION;

	END_CASE

	pKuka.convert.ValuesToPosition();
	pKuka.convert.ValuesToCOORDSYS.Base := pKuka.convert.ValuesToPosition.baseNo;
	pKuka.convert.ValuesToCOORDSYS.IPO_Mode := 0; // #BASE
	pKuka.convert.ValuesToCOORDSYS();

	pKuka.tempPosition := pKuka.convert.ValuesToPosition.outputPos;

	pKuka.motion.KRC_MoveDirectAbsolute.CoordinateSystem := pKuka.convert.ValuesToCOORDSYS.COORDSYS;
	pKuka.motion.KRC_MoveDirectAbsolute.Position := pKuka.tempPosition;

	pKuka.motion.KRC_MoveDirectAbsolute.ExecuteCmd := TRUE;
	IF pKuka.motion.KRC_MoveDirectAbsolute.Done THEN
		pKuka.motion.KRC_MoveDirectAbsolute.ExecuteCmd := FALSE;
		robotDone[i] := FALSE;
		cm.state := 1000;
	END_IF

END_ACTION
```

#### RobotAssembly.st
```iecst
ACTION RobotAssembly:

	CASE cm.state OF

		1000:
			cm.description := 'Define order-specific approach point at magazine';

			IF robotExecute[i] THEN
				cm.state := 1010;

				robotBusy[i] := TRUE;
				pKuka.convert.ValuesToPosition.posType := APPROACH_MAGAZINE;
				pKuka.convert.ValuesToPosition();

				pKuka.tempPosition := pKuka.convert.ValuesToPosition.outputPos;

				// The following order-specific adjustments are possible since we at this point know that the robot has returned to home position (main approach point) in cm.state = 500
				CASE pKuka.axisGroupIdx OF
					1:
						CASE orderSpec[i] OF
							1: // Black cover
								pKuka.tempPosition.X := pKuka.tempPosition.X; // Change when ready

							2: // White cover
								pKuka.tempPosition.X := pKuka.tempPosition.X - 80; // Change when ready

							3: // Blue cover
								pKuka.tempPosition.X := pKuka.tempPosition.X - 160; // Change when ready
						END_CASE

					3:
						// Do Nothing
						cm.state := 1020;

					4:
						CASE orderSpec[i] OF
							1: // 1 fuse
								pKuka.tempPosition.X := pKuka.tempPosition.X + fusePickOffset;
								fusePickOffset := fusePickOffset * (-1); // Change pick side

							2: // 2 fuses
								pKuka.tempPosition.X := pKuka.tempPosition.X; // Change when ready
						END_CASE

					5:
						CASE orderSpec[i] OF
							1: // Black cover
								pKuka.tempPosition.X := pKuka.tempPosition.X; // Change when ready

							2: // White cover
								pKuka.tempPosition.X := pKuka.tempPosition.X + 80; // Change when ready

							3: // Blue cover
								pKuka.tempPosition.X := pKuka.tempPosition.X + 160; // Change when ready
						END_CASE

				END_CASE
			END_IF

		1010:
			cm.description := 'Move to order-specific approach point at magazine';
			pKuka.convert.ValuesToCOORDSYS.IPO_Mode := 0; // #BASE
			pKuka.convert.ValuesToCOORDSYS();

			pKuka.motion.KRC_MoveDirectAbsolute.CoordinateSystem := pKuka.convert.ValuesToCOORDSYS.COORDSYS;

			pKuka.motion.KRC_MoveDirectAbsolute.Position := pKuka.tempPosition;

			pKuka.motion.KRC_MoveDirectAbsolute.ExecuteCmd := TRUE;
			IF pKuka.motion.KRC_MoveDirectAbsolute.Done THEN
				pKuka.motion.KRC_MoveDirectAbsolute.ExecuteCmd := FALSE;
				cm.state := 1020;
			END_IF

		1020:
			cm.description := 'Move to pickup point with relative linear movement';

			pKuka.convert.ValuesToCOORDSYS.IPO_Mode := 1; // #TOOL
			pKuka.convert.ValuesToCOORDSYS();

			pKuka.motion.KRC_MoveLinearRelative.CoordinateSystem := pKuka.convert.ValuesToCOORDSYS.COORDSYS;

			pKuka.tempPosition.X := pKuka.tempPosition.Y := pKuka.tempPosition.Z := pKuka.tempPosition.A := pKuka.tempPosition.B := pKuka.tempPosition.C
			:= 0;
			pKuka.tempPosition.Z := -relativeDistance;
			// Status and turn is already set from moving to approach point

			pKuka.motion.KRC_MoveLinearRelative.Position := pKuka.tempPosition;

			pKuka.motion.KRC_MoveLinearRelative.ExecuteCmd := TRUE;
			IF pKuka.motion.KRC_MoveLinearRelative.Done THEN
				pKuka.motion.KRC_MoveLinearRelative.ExecuteCmd := FALSE;
				cm.state := 1030;
			END_IF

		1030:
			cm.description := 'Close gripper and wait a little before moving to ensure proper grip';

			pKuka.gripperAction.action := CLOSE;

			pKuka.TON.PT := REAL_TO_TIME(gripperWaitTime); // in ms
			pKuka.TON.IN := TRUE;
			IF pKuka.TON.Q THEN
				pKuka.TON.IN := FALSE;
				cm.state := 1040;
			END_IF

		1040:
			cm.description := 'Move to approach point with relative linear movement';

			pKuka.tempPosition.X := pKuka.tempPosition.Y := pKuka.tempPosition.Z := pKuka.tempPosition.A := pKuka.tempPosition.B := pKuka.tempPosition.C
			:= 0;
			pKuka.tempPosition.Z := relativeDistance;
			// Status and turn is already set from moving to approach point

			pKuka.motion.KRC_MoveLinearRelative.Position := pKuka.tempPosition;

			pKuka.motion.KRC_MoveLinearRelative.ExecuteCmd := TRUE;
			IF pKuka.motion.KRC_MoveLinearRelative.Done THEN
				pKuka.motion.KRC_MoveLinearRelative.ExecuteCmd := FALSE;
				cm.state := 1050;
			END_IF

		1050:
			cm.description := 'Move to approach point of workstation with absolute linear movement';

			pKuka.convert.ValuesToPosition.posType := APPROACH_WORKSTATION;
			pKuka.convert.ValuesToPosition();

			pKuka.convert.ValuesToCOORDSYS.Base := pKuka.convert.ValuesToPosition.baseNo; // ACOPOS6D frame
			pKuka.convert.ValuesToCOORDSYS.IPO_Mode := 0; // #BASE
			pKuka.convert.ValuesToCOORDSYS();

			pKuka.tempPosition := pKuka.convert.ValuesToPosition.outputPos;

			pKuka.motion.KRC_MoveDirectAbsolute.CoordinateSystem := pKuka.convert.ValuesToCOORDSYS.COORDSYS;
			pKuka.motion.KRC_MoveDirectAbsolute.Position := pKuka.tempPosition;

			pKuka.motion.KRC_MoveDirectAbsolute.ExecuteCmd := TRUE;
			IF pKuka.motion.KRC_MoveDirectAbsolute.Done THEN
				pKuka.motion.KRC_MoveDirectAbsolute.ExecuteCmd := FALSE;
				cm.state := 1060;
			END_IF

		1060:
			cm.description := 'Move to placement point at workstation with relative linear movement';

			pKuka.convert.ValuesToCOORDSYS.IPO_Mode := 1; // #TOOL
			pKuka.convert.ValuesToCOORDSYS();

			pKuka.motion.KRC_MoveLinearRelative.CoordinateSystem := pKuka.convert.ValuesToCOORDSYS.COORDSYS;

			pKuka.tempPosition.X := pKuka.tempPosition.Y := pKuka.tempPosition.Z := pKuka.tempPosition.A := pKuka.tempPosition.B := pKuka.tempPosition.C
			:= 0;
			pKuka.tempPosition.Z := -relativeDistance; // Move 100 mm forwards to placement position
			// Status and turn is already set from moving to approach point

			pKuka.motion.KRC_MoveLinearRelative.Position := pKuka.tempPosition;

			pKuka.motion.KRC_MoveLinearRelative.ExecuteCmd := TRUE;
			IF pKuka.motion.KRC_MoveLinearRelative.Done THEN
				pKuka.motion.KRC_MoveLinearRelative.ExecuteCmd := FALSE;
				cm.state := 1070;
			END_IF

		1070:
			cm.description := 'Open gripper and wait a little before moving to ensure proper grip';

			pKuka.gripperAction.action := OPEN;

			pKuka.TON.PT := REAL_TO_TIME(gripperWaitTime); // in ms
			pKuka.TON.IN := TRUE;
			IF pKuka.TON.Q THEN
				pKuka.TON.IN := FALSE;
				cm.state := 1080;
			END_IF

		1080:
			cm.description := 'Move back to approach point at workstation with relative linear movement';

			pKuka.convert.ValuesToCOORDSYS.IPO_Mode := 1; // #TOOL
			pKuka.convert.ValuesToCOORDSYS();

			pKuka.motion.KRC_MoveLinearRelative.CoordinateSystem := pKuka.convert.ValuesToCOORDSYS.COORDSYS;

			pKuka.tempPosition.X := pKuka.tempPosition.Y := pKuka.tempPosition.Z := pKuka.tempPosition.A := pKuka.tempPosition.B := pKuka.tempPosition.C
			:= 0;
			pKuka.tempPosition.Z := relativeDistance;
			// Status and turn is already set from moving to approach point

			pKuka.motion.KRC_MoveLinearRelative.Position := pKuka.tempPosition;

			pKuka.motion.KRC_MoveLinearRelative.ExecuteCmd := TRUE;
			IF pKuka.motion.KRC_MoveLinearRelative.Done THEN
				pKuka.motion.KRC_MoveLinearRelative.ExecuteCmd := FALSE;
				robotDone[i] := TRUE;
				cm.state := 1090;
			END_IF

		1090:
			cm.description := 'Move back to home position';
			RobotHoming;

	END_CASE

END_ACTION
```

#### RobotProcess.st
```iecst
ACTION RobotProcess:

	CASE cm.state OF

		1000:
			cm.description := 'Define order-specific approach point at magazine';

			IF robotExecute[i] THEN
				robotBusy[i] := TRUE;
				pKuka.convert.ValuesToPosition.posType := APPROACH_WORKSTATION;
				pKuka.convert.ValuesToPosition();

				pKuka.tempPosition := pKuka.convert.ValuesToPosition.outputPos;

				CASE pKuka.axisGroupIdx OF
					2: //Drilling robot
						// Seen from ACOPOS 6D frame: Bottom right -> bottom left -> top left -> top right

						CASE numDoneHoles OF
							0: // Simply default approach position

							1:
								pKuka.tempPosition.X := pKuka.tempPosition.X - drillXOffset;
								pKuka.tempPosition.Status := 2; // 010
								pKuka.tempPosition.Turn := 35; // 100011

							2:
								pKuka.tempPosition.X := pKuka.tempPosition.X - drillXOffset;
								pKuka.tempPosition.Y := pKuka.tempPosition.Y + drillYOffset;
								pKuka.tempPosition.Status := 6; // 110
								pKuka.tempPosition.Turn := 51; // 110011

							3:
								pKuka.tempPosition.Y := pKuka.tempPosition.Y + drillYOffset;
								pKuka.tempPosition.Status := 6; // 110
								pKuka.tempPosition.Turn := 51; // 110011

						END_CASE

				END_CASE

				cm.state := 1010;

			END_IF

		1010:
			cm.description := 'Move to order-specific approach point';

			pKuka.convert.ValuesToCOORDSYS.Base := pKuka.convert.ValuesToPosition.baseNo;
			pKuka.convert.ValuesToCOORDSYS.IPO_Mode := 0; // #BASE
			pKuka.convert.ValuesToCOORDSYS();

			pKuka.motion.KRC_MoveDirectAbsolute.CoordinateSystem := pKuka.convert.ValuesToCOORDSYS.COORDSYS;

			pKuka.motion.KRC_MoveDirectAbsolute.Position := pKuka.tempPosition;

			pKuka.motion.KRC_MoveDirectAbsolute.ExecuteCmd := TRUE;
			IF pKuka.motion.KRC_MoveDirectAbsolute.Done THEN
				pKuka.motion.KRC_MoveDirectAbsolute.ExecuteCmd := FALSE;
				cm.state := 1020;
			END_IF

		1020:
			cm.description := 'Perform order-specific motion with relative linear movement';

			// Relative movement w.r.t tool does not require defining base
			pKuka.convert.ValuesToCOORDSYS.IPO_Mode := 1; // #TOOL
			pKuka.convert.ValuesToCOORDSYS();

			pKuka.motion.KRC_MoveLinearRelative.CoordinateSystem := pKuka.convert.ValuesToCOORDSYS.COORDSYS;

			pKuka.tempPosition.X := pKuka.tempPosition.Y := pKuka.tempPosition.Z := pKuka.tempPosition.A := pKuka.tempPosition.B := pKuka.tempPosition.C
			:= 0;
			CASE pKuka.axisGroupIdx OF
				2: pKuka.tempPosition.Z := -(relativeDrillDistance + 6);
			END_CASE
			// Status and turn is already set from moving to approach point

			pKuka.motion.KRC_MoveLinearRelative.Position := pKuka.tempPosition;

			pKuka.motion.KRC_MoveLinearRelative.ExecuteCmd := TRUE;
			IF pKuka.motion.KRC_MoveLinearRelative.Done THEN
				pKuka.motion.KRC_MoveLinearRelative.ExecuteCmd := FALSE;
				cm.state := 1030;
			END_IF

		1030:

			cm.description := 'Move back to approach point with relative linear movement';

			pKuka.convert.ValuesToCOORDSYS.IPO_Mode := 1; // #TOOL
			pKuka.convert.ValuesToCOORDSYS();

			pKuka.motion.KRC_MoveLinearRelative.CoordinateSystem := pKuka.convert.ValuesToCOORDSYS.COORDSYS;

			pKuka.tempPosition.X := pKuka.tempPosition.Y := pKuka.tempPosition.A := pKuka.tempPosition.B := pKuka.tempPosition.C
			:= 0;
			pKuka.tempPosition.Z := -1*pKuka.tempPosition.Z; // go back
			// Status and turn is already set from moving to approach point

			pKuka.motion.KRC_MoveLinearRelative.Position := pKuka.tempPosition;

			pKuka.motion.KRC_MoveLinearRelative.ExecuteCmd := TRUE;
			IF pKuka.motion.KRC_MoveLinearRelative.Done THEN
				pKuka.motion.KRC_MoveLinearRelative.ExecuteCmd := FALSE;

				CASE pKuka.axisGroupIdx OF
					2: //Drilling robot
						numDoneHoles := numDoneHoles + 1;

						// Check if more holes are needed for the specific order
						IF numDoneHoles < orderSpec[i] THEN
							// Define next order-specific approach point
							cm.state := 1000;
						ELSE
							// Order is completed, we move back to mint approach point (APPROACH_WORKSTATION)
							numDoneHoles := 0;
							robotDone[i] := TRUE;
							cm.state := 1040;
						END_IF
				END_CASE

			END_IF

		1040:
			cm.description := 'Move back to home position';

			RobotHoming;

	END_CASE

END_ACTION
```

#### JointMovement.st
```iecst
ACTION JointMovement:

	CASE pKuka.cm.state OF

		0:
			// Set initial parameters for movement
			pKuka.motion.KRC_MoveAxisAbsolute.ExecuteCmd 			:= FALSE;
			pKuka.motion.KRC_MoveAxisAbsolute.AxisGroupIdx 			:= pKuka.axisGroupIdx;
			pKuka.motion.KRC_MoveAxisAbsolute.KRC_AxisGroupRefArr	:= ADR(AxisRef);
			pKuka.motion.KRC_MoveAxisAbsolute.Velocity 				:= 10;
			pKuka.motion.KRC_MoveAxisAbsolute.Acceleration 			:= 20;
			pKuka.motion.KRC_MoveAxisAbsolute.BufferMode 			:= 2;

			position1.A1 := 0;
			position1.A2 := -70;
			position1.A3 := 90;
			position1.A4 := 0;
			position1.A5 := -90;
			position1.A6 := 0;

			position2.A1 := 0;
			position2.A2 := -90;
			position2.A3 := 90;
			position2.A4 := 0;
			position2.A5 := 80;
			position2.A6 := 0;

			pKuka.cm.state := 10;

		10: // Set initial position
			pKuka.motion.KRC_MoveAxisAbsolute.AxisPosition := position1;

			pKuka.motion.KRC_MoveAxisAbsolute.ExecuteCmd 	:= TRUE;
			IF pKuka.motion.KRC_MoveAxisAbsolute.Done THEN
				pKuka.motion.KRC_MoveAxisAbsolute.ExecuteCmd := FALSE;
				pKuka.cm.state := 20;
			END_IF

		20:	// Set second position
			pKuka.motion.KRC_MoveAxisAbsolute.AxisPosition := position2;

			pKuka.motion.KRC_MoveAxisAbsolute.ExecuteCmd	:= TRUE;
			IF pKuka.motion.KRC_MoveAxisAbsolute.Done THEN
				pKuka.motion.KRC_MoveAxisAbsolute.ExecuteCmd	:= FALSE;
				pKuka.cm.state := 10;
			END_IF

	END_CASE

	pKuka.motion.KRC_MoveAxisAbsolute();

END_ACTION
```

#### LinearMovement.st
```iecst
ACTION LinearMovement:

	CASE pKuka.cm.state OF

		0:
			//Set frames as coordsys
			mxa_ValuesToCOORDSYS_0.Tool 	:= 1; // Change to 1 when it works
			mxa_ValuesToCOORDSYS_0.Base 	:= 1;
			mxa_ValuesToCOORDSYS_0.IPO_Mode := 0;

			pKuka.cm.state := 10;

		10:
			coordSys := mxa_ValuesToCOORDSYS_0.COORDSYS;

			pKuka.motion.KRC_MoveLinearAbsolute.AxisGroupIdx 		:= pKuka.axisGroupIdx;
			pKuka.motion.KRC_MoveLinearAbsolute.KRC_AxisGroupRefArr	:= ADR(AxisRef);
			pKuka.motion.KRC_MoveLinearAbsolute.Velocity			:= 10;
			pKuka.motion.KRC_MoveLinearAbsolute.Acceleration  		:= 20;
			pKuka.motion.KRC_MoveLinearAbsolute.CoordinateSystem	:= coordSys;
			pKuka.motion.KRC_MoveLinearAbsolute.OriType 			:= 0;
			pKuka.motion.KRC_MoveLinearAbsolute.BufferMode			:= 2;

			pKuka.cm.state := 20;

		20:
			endPOS.X := 302;
			endPOS.Y := -2;
			endPOS.Z := 527;
			endPOS.A := -178;
			endPOS.B := 26;
			endPOS.C := -178;
			endPOS.Status := 2; //010
			endPOS.Turn := 2; //000010

			pKuka.motion.KRC_MoveLinearAbsolute.Position		:= endPOS;

			pKuka.motion.KRC_MoveLinearAbsolute.ExecuteCmd 		:= TRUE;
			IF pKuka.motion.KRC_MoveLinearAbsolute.Done THEN
				pKuka.motion.KRC_MoveLinearAbsolute.ExecuteCmd 	:= FALSE;
				pKuka.cm.state := 30;
			END_IF

		30:
			endPOS.X := 430;
			endPOS.Y := -2;
			endPOS.Z := 527;
			endPOS.A := -178;
			endPOS.B := 26;
			endPOS.C := -178;
			endPOS.Status := 2; //010
			endPOS.Turn := 2; //000010

			pKuka.motion.KRC_MoveLinearAbsolute.Position		:= endPOS;

			pKuka.motion.KRC_MoveLinearAbsolute.ExecuteCmd 		:= TRUE;
			IF pKuka.motion.KRC_MoveLinearAbsolute.Done THEN
				pKuka.motion.KRC_MoveLinearAbsolute.ExecuteCmd 	:= FALSE;
				pKuka.cm.state 	:= 20;
			END_IF

	END_CASE

	mxa_ValuesToCOORDSYS_0();
	pKuka.motion.KRC_MoveLinearAbsolute();

END_ACTION
```

#### LocalFunctions.fun
```iecst
{REDUND_OK} FUNCTION_BLOCK GripperAction (*TODO: Add your comment here*) (*$GROUP=User,$CAT=User,$GROUPICON=User.png,$CATICON=User.png*)
	VAR_INPUT
		whitePin : REFERENCE TO BOOL;
		blackPin : REFERENCE TO BOOL;
		action : gripper_action_type;
	END_VAR
END_FUNCTION_BLOCK

{REDUND_ERROR} FUNCTION_BLOCK ValuesToMagazineFrame (*TODO: Add your comment here*) (*$GROUP=User,$CAT=User,$GROUPICON=User.png,$CATICON=User.png*)
	VAR_INPUT
		axisGroupIdx : USINT;
	END_VAR
	VAR_OUTPUT
		outputFrame : FRAME;
	END_VAR
END_FUNCTION_BLOCK

{REDUND_ERROR} FUNCTION_BLOCK ValuesToPosition (*TODO: Add your comment here*) (*$GROUP=User,$CAT=User,$GROUPICON=User.png,$CATICON=User.png*)
	VAR_INPUT
		axisGroupIdx : {REDUND_UNREPLICABLE} USINT;
		posType : robot_position_type;
	END_VAR
	VAR_OUTPUT
		outputPos : E6POS;
		baseNo : USINT;
	END_VAR
	VAR
		ValuesToCorrection_0 : ValuesToCorrection;
	END_VAR
END_FUNCTION_BLOCK

{REDUND_ERROR} {REDUND_UNREPLICABLE} FUNCTION_BLOCK EETypeToFrame (*TODO: Add your comment here*) (*$GROUP=User,$CAT=User,$GROUPICON=User.png,$CATICON=User.png*)
	VAR_INPUT
		eeType : {REDUND_UNREPLICABLE} end_effector_type;
	END_VAR
	VAR_OUTPUT
		frame : {REDUND_UNREPLICABLE} FRAME;
	END_VAR
	VAR CONSTANT
		SchunkLength : REAL := 72.7+2*3.2;
	END_VAR
END_FUNCTION_BLOCK

{REDUND_ERROR} FUNCTION_BLOCK ValuesToCorrection (*TODO: Add your comment here*) (*$GROUP=User,$CAT=User,$GROUPICON=User.png,$CATICON=User.png*)
	VAR_INPUT
		robotIdx : USINT;
		baseNo : USINT;
	END_VAR
	VAR_OUTPUT
		posCorrections : E6POS;
	END_VAR
END_FUNCTION_BLOCK
```

#### EETypeToFrame.st
```iecst
(* TODO: Add your comment here *)
FUNCTION_BLOCK EETypeToFrame

	frame.X := 0;
	frame.Y := 0;
	frame.Z := SchunkLength; //79.1 (with base plate)
	frame.A := 0;
	frame.B := 0;
	frame.C := 0;

	CASE eeType OF

		COVER_EE:

			frame.Z := frame.Z + 29.40; // Change when we know

		DRILL_EE:
			frame.Z := frame.Z; // Change when we know

		PCB_EE:
			frame.Z := frame.Z + 25.11;
			//frame.C := 180;

		FUSE_EE:
			frame.Z := frame.Z + 20; // Change when we know

	END_CASE

END_FUNCTION_BLOCK
```

#### ValuesToPosition.st
```iecst
// DEFAULT is 0, -120, 120, 0, 90, 0 in joint angles (without tool - remember to add tool for nice configuration)

// DEFAULT is with reference to WORLD frame
// APPROACH_MAGAZINE is with reference to its own magazine frame
// APPROACH_WORKSTATION is with reference to ACOPOS6D frame

FUNCTION_BLOCK ValuesToPosition
	CASE axisGroupIdx OF
		///////////////// ROBOT 1 /////////////////
		1:
			CASE posType OF
				DEFAULT:
					outputPos.X := 915;
					outputPos.Y := 120;
					outputPos.Z := 536.147;
					outputPos.A := 0;
					outputPos.B := 0;
					outputPos.C := 180;
					outputPos.Status := 2; // 010
					outputPos.Turn := 2; // 000010

					baseNo := 0;

				APPROACH_MAGAZINE:
					outputPos.X := 200.000;
					outputPos.Y := 203.066;
					outputPos.Z := 157.556;
					outputPos.A := 0;
					outputPos.B := 0;
					outputPos.C := 135;
					outputPos.Status := 2; // 010 Third bit is different from manual
					outputPos.Turn := 10; // 001010

					baseNo := 2;

				APPROACH_WORKSTATION:
					outputPos.X := 660;
					outputPos.Y := 60;
					outputPos.Z := (1 + 9.85 + 5) + relativeDistance + 2;
					outputPos.A := 0;
					outputPos.B := 0;
					outputPos.C := 180;
					outputPos.Status := 2; // 010
					outputPos.Turn := 2; // 000010

					baseNo := 1;

			END_CASE

		///////////////////////////////////////////

		///////////////// ROBOT 2 /////////////////
		2:
			CASE posType OF
				DEFAULT:
					outputPos.X := 930;
					outputPos.Y := 840;
					outputPos.Z := 525.167;
					outputPos.A := 0;
					outputPos.B := 0;
					outputPos.C := 180;
					outputPos.Status := 2; // 010
					outputPos.Turn := 2; // 000010

					baseNo := 0;

				APPROACH_WORKSTATION:
					outputPos.X := 660 + 27; //Last term is x offset of bottom right hole
					outputPos.Y := 420 - 53; //Last term is y offset of bottom right hole
					outputPos.Z := (1 + 9.85 + 5 + 13) + relativeDistance + 100; // Remember to change
					outputPos.A := 0;
					outputPos.B := 0;
					outputPos.C := 180;
					outputPos.Status := 2; // 010
					outputPos.Turn := 35; // 100011

					baseNo := 1;

			END_CASE

		///////////////////////////////////////////

		///////////////// ROBOT 3 /////////////////
		3:
			CASE posType OF
				DEFAULT:
					outputPos.X := 930;
					outputPos.Y := 1320;
					outputPos.Z := 525.167;
					outputPos.A := 0;
					outputPos.B := 0;
					outputPos.C := 180;
					outputPos.Status := 2; // 010
					outputPos.Turn := 2; // 000010

					baseNo := 0;

				APPROACH_MAGAZINE:
					outputPos.X := 152.740;
					outputPos.Y := 219.477;
					outputPos.Z := 148.927;
					outputPos.A := -90.000;
					outputPos.B := -45.000;
					outputPos.C := -180.000;
					outputPos.Status := 2; // 010
					outputPos.Turn := 3; // 000011

					baseNo := 2;

				APPROACH_WORKSTATION:
					outputPos.X := 660;
					outputPos.Y := 780 + 32.79; // 32.79 represents shift from center to fuse bracket
					outputPos.Z := (1 + 9.85 + 5 + 6.7 + 1.5 + 2) + relativeDistance + 2;
					outputPos.A := 0;
					outputPos.B := 0;
					outputPos.C := 180;
					outputPos.Status := 2; // 010
					outputPos.Turn := 35; // 100011

					baseNo := 1;

			END_CASE

		///////////////////////////////////////////

		///////////////// ROBOT 4 /////////////////
		4:
			CASE posType OF
				DEFAULT:
					outputPos.X := 270;
					outputPos.Y := 1320;
					outputPos.Z := 525.167;
					outputPos.A := -180;
					outputPos.B := 0;
					outputPos.C := 180;
					outputPos.Status := 2; // 010
					outputPos.Turn := 2; // 000010

					baseNo := 0;

				APPROACH_MAGAZINE:
					outputPos.X := 120;
					outputPos.Y := 250.263;
					outputPos.Z := 196.383;
					outputPos.A := 0;
					outputPos.B := 0;
					outputPos.C := 135;
					outputPos.Status := 2; // 010
					outputPos.Turn := 10; // 001010

					baseNo := 2;

				APPROACH_WORKSTATION:
					outputPos.X := 60;
					outputPos.Y := 780 + 32.79; // 32.79 represents shift from center to fuse bracket
					outputPos.Z := (1 + 9.85 + 5 + 6.7 + 1.5 + 2 + 0.5) + relativeDistance;
					outputPos.A := 90;
					outputPos.B := 0;
					outputPos.C := 180;
					outputPos.Status := 2; // 010
					outputPos.Turn := 34; // 100010

					baseNo := 1;

			END_CASE

		///////////////////////////////////////////

		///////////////// ROBOT 5 /////////////////
		5:
			CASE posType OF
				DEFAULT:
					outputPos.X := 270;
					outputPos.Y := 840;
					outputPos.Z := 525.167;
					outputPos.A := -180;
					outputPos.B := 0;
					outputPos.C := 180;
					outputPos.Status := 2; // 010
					outputPos.Turn := 2; // 000010

					baseNo := 0;

				APPROACH_MAGAZINE:
					outputPos.X := 40;
					outputPos.Y := 203.067;
					outputPos.Z := 157.557;
					outputPos.A := 0;
					outputPos.B := 0;
					outputPos.C := 135;
					outputPos.Status := 2; // 010
					outputPos.Turn := 2; // 000010

					baseNo := 2;

				APPROACH_WORKSTATION:
					outputPos.X := 60;
					outputPos.Y := 420;
					outputPos.Z := (1 + 9.85 + 5 + 13) + relativeDistance;
					outputPos.A := -180;
					outputPos.B := 0;
					outputPos.C := 180;
					outputPos.Status := 2; // 010
					outputPos.Turn := 2; // 000010

					baseNo := 1;

			END_CASE

		///////////////////////////////////////////

		///////////////// ROBOT 6 /////////////////
		6:
			CASE posType OF
				DEFAULT:
					outputPos.X := 285;
					outputPos.Y := 120;
					outputPos.Z := 536.147;
					outputPos.A := -180;
					outputPos.B := 0;
					outputPos.C := 180;
					outputPos.Status := 2; // 010
					outputPos.Turn := 2; // 000010

					baseNo := 0;

				APPROACH_MAGAZINE:
					outputPos.X := -60;
					outputPos.Y := 160;
					outputPos.Z := 290;
					outputPos.A := -180;
					outputPos.B := 0;
					outputPos.C := 180;
					outputPos.Status := 2; // 010
					outputPos.Turn := 35; // 100011

					baseNo := 2;

				APPROACH_WORKSTATION:
					outputPos.X := 60;
					outputPos.Y := 60;
					outputPos.Z := (1 + 9.85 + 5) + relativeDistance + 2;
					outputPos.A := -180;
					outputPos.B := 0;
					outputPos.C := 180;
					outputPos.Status := 2; // 010
					outputPos.Turn := 35; // 100011

					baseNo := 1;

			END_CASE

	END_CASE

	ValuesToCorrection_0.baseNo := baseNo;
	ValuesToCorrection_0.robotIdx := axisGroupIdx;
	ValuesToCorrection_0();

	outputPos.X := outputPos.X + ValuesToCorrection_0.posCorrections.X;
	outputPos.Y := outputPos.Y + ValuesToCorrection_0.posCorrections.Y;
	outputPos.Z := outputPos.Z + ValuesToCorrection_0.posCorrections.Z;
	outputPos.A := outputPos.A + ValuesToCorrection_0.posCorrections.A;
	outputPos.B := outputPos.B + ValuesToCorrection_0.posCorrections.B;
	outputPos.C := outputPos.C + ValuesToCorrection_0.posCorrections.C;

END_FUNCTION_BLOCK
```

#### ValuesToMagazineFrame.st
```iecst
(* TODO: Add your comment here *)
FUNCTION_BLOCK ValuesToMagazineFrame

	outputFrame.X := 0;
	outputFrame.Y := 0;
	outputFrame.Z := 0;
	outputFrame.A := 0;
	outputFrame.B := 0;
	outputFrame.C := 0;

	CASE axisGroupIdx OF
		1: // Bottom cover magazine frame
			outputFrame.X := 600;
			outputFrame.Y := 0;
			outputFrame.Z := 6.3;
			outputFrame.A := 0;
			outputFrame.B := 0;
			outputFrame.C := 0;

		2: // DRILLING HAS NO MAGAZINE

		3: // PCB magazine frame
			outputFrame.X := 840;
			outputFrame.Y := 1440;
			outputFrame.Z := 6.3;
			outputFrame.A := 180;
			outputFrame.B := 0;
			outputFrame.C := 0;

		4: // Fuse magazine frame
			outputFrame.X := 600;
			outputFrame.Y := 1440;
			outputFrame.Z := 0;
			outputFrame.A := 180;
			outputFrame.B := 0;
			outputFrame.C := 0;

		5: // Top cover magazine frame
			outputFrame.X := 0;
			outputFrame.Y := 720;
			outputFrame.Z := 0;
			outputFrame.A := -90;
			outputFrame.B := 0;
			outputFrame.C := 0;

		6: // Unloading frame
			outputFrame.X := 360;
			outputFrame.Y := 0;
			outputFrame.Z := 0;
			outputFrame.A := 0;
			outputFrame.B := 0;
			outputFrame.C := 0;

	END_CASE

END_FUNCTION_BLOCK
```

#### ValuesToCorrection.st
```iecst
(* TODO: Add your comment here *)
FUNCTION_BLOCK ValuesToCorrection

	posCorrections.X := 0;
	posCorrections.Y := 0;
	posCorrections.Z := 0;
	posCorrections.A := 0;
	posCorrections.B := 0;
	posCorrections.C := 0;

	CASE robotIdx OF

		1:
			CASE baseNo OF
				0: // w.r.t world frame

				1: // w.r.t acopos frame
					posCorrections.Y := 1.5;

				2: // w.r.t magazine frame
					posCorrections.X := -4;
					posCorrections.Y := 2;
					posCorrections.Z := 2;
			END_CASE
		2:

		3:
			CASE baseNo OF
				0: // w.r.t world frame

				1: // w.r.t acopos frame
					posCorrections.X := 2;
					posCorrections.Y := -0.2;

				2: // w.r.t magazine frame
					posCorrections.X := 1;
					posCorrections.Y := 0.5;
					posCorrections.Z := -0.5;
			END_CASE

		4:
			CASE baseNo OF
				0: // w.r.t world frame

				1: // w.r.t acopos frame
					posCorrections.X := -1;
					posCorrections.Y := -0.3;

				2: // w.r.t magazine frame
					posCorrections.X := 0.85;
					posCorrections.Y := 0;
					posCorrections.Z := 4.0;

			END_CASE
		5:
			CASE baseNo OF
				0: // w.r.t world frame

				1: // w.r.t acopos frame
					posCorrections.X := -0.5;
					posCorrections.Y := 3;
					posCorrections.Z := -6;

				2: // w.r.t magazine frame
					posCorrections.X := 2;
					posCorrections.Y := -5;
					posCorrections.Z := 9;

			END_CASE
		6:

	END_CASE

END_FUNCTION_BLOCK
```

#### KUKABottomCover.st - not listed in the package file held
```iecst
ACTION KUKABottomCover:

	CASE cm.state OF

		1000:
			cm.description := 'Initialising parameters';

			pKuka.convert.ValuesToCOORDSYS.Tool := 1;
			pKuka.convert.ValuesToCOORDSYS();

			pKuka.convert.ValuesToPosition.axisGroupIdx := pKuka.axisGroupIdx;
			pKuka.convert.ValuesToPosition();

			pKuka.motion.KRC_MoveDirectAbsolute.AxisGroupIdx := pKuka.motion.KRC_MoveLinearAbsolute.AxisGroupIdx := pKuka.motion.KRC_MoveLinearRelative.AxisGroupIdx
				:=  pKuka.axisGroupIdx;
			pKuka.motion.KRC_MoveDirectAbsolute.KRC_AxisGroupRefArr := pKuka.motion.KRC_MoveLinearAbsolute.KRC_AxisGroupRefArr := pKuka.motion.KRC_MoveLinearRelative.KRC_AxisGroupRefArr
				:= ADR(AxisRef);
			pKuka.motion.KRC_MoveDirectAbsolute.Velocity := pKuka.motion.KRC_MoveLinearAbsolute.Velocity := pKuka.motion.KRC_MoveLinearRelative.Velocity
				:= 5; // Velocity in percent
			pKuka.motion.KRC_MoveDirectAbsolute.Acceleration := pKuka.motion.KRC_MoveLinearAbsolute.Acceleration := pKuka.motion.KRC_MoveLinearRelative.Acceleration
				:= 20; // Acceleration in percent
			pKuka.motion.KRC_MoveDirectAbsolute.BufferMode := pKuka.motion.KRC_MoveLinearAbsolute.BufferMode := pKuka.motion.KRC_MoveLinearRelative.BufferMode
				:= 2; // BUFFERED
			pKuka.motion.KRC_MoveLinearAbsolute.OriType := pKuka.motion.KRC_MoveLinearRelative.OriType
				:= 0; // 0: VAR | 1: CONSTANT | 2: JOINT
			pKuka.motion.KRC_MoveDirectAbsolute.ExecuteCmd := pKuka.motion.KRC_MoveLinearAbsolute.ExecuteCmd := pKuka.motion.KRC_MoveLinearRelative.ExecuteCmd
				:= FALSE;

			cm.state := 1010;

		1010:
			cm.description := 'Waiting for flag to start movement';

			IF robotOperating[i] THEN
				cm.state := 1020;
			END_IF

		1020:
			cm.description := 'Move to approach point of magazine with absolute joint movement';

			pKuka.convert.ValuesToCOORDSYS.Base := 2; // Magazine frame
			pKuka.convert.ValuesToCOORDSYS.IPO_Mode := 0; // #BASE
			pKuka.convert.ValuesToCOORDSYS();

			pKuka.convert.ValuesToPosition.posType := APPROACH_MAGAZINE;
			pKuka.convert.ValuesToPosition();

			pKuka.tempPosition := pKuka.convert.ValuesToPosition.outputPos;

			// Fit the position with the specified cover type
			CASE orderSpec[i] OF
				0: // Black cover
					pKuka.tempPosition.X := pKuka.tempPosition.X + 0; // Change when ready

				1: // White cover
					pKuka.tempPosition.X := pKuka.tempPosition.X + 80; // Change when ready

				2: // Blue cover
					pKuka.tempPosition.X := pKuka.tempPosition.X + 160; // Change when ready

			END_CASE

			pKuka.motion.KRC_MoveDirectAbsolute.CoordinateSystem := pKuka.convert.ValuesToCOORDSYS.COORDSYS;
			pKuka.motion.KRC_MoveDirectAbsolute.Position := pKuka.tempPosition;

			pKuka.motion.KRC_MoveDirectAbsolute.ExecuteCmd := TRUE;
			IF pKuka.motion.KRC_MoveDirectAbsolute.Done THEN
				pKuka.motion.KRC_MoveDirectAbsolute.ExecuteCmd := FALSE;
				cm.state := 1030;
			END_IF

		1030:
			cm.description := 'Move to pickup point at magazine with relative linear movement';

			pKuka.convert.ValuesToCOORDSYS.IPO_Mode := 1; // #TOOL
			pKuka.convert.ValuesToCOORDSYS();

			pKuka.motion.KRC_MoveLinearRelative.CoordinateSystem := pKuka.convert.ValuesToCOORDSYS.COORDSYS;

			pKuka.tempPosition.X := pKuka.tempPosition.Y := pKuka.tempPosition.Z := pKuka.tempPosition.A := pKuka.tempPosition.B := pKuka.tempPosition.C
				:= 0;
			pKuka.tempPosition.Z := 45; // Move 100 mm forwards to pickup position
			// Status and turn is already set from moving to approach point

			pKuka.motion.KRC_MoveLinearRelative.Position := pKuka.tempPosition;

			pKuka.motion.KRC_MoveLinearRelative.ExecuteCmd := TRUE;
			IF pKuka.motion.KRC_MoveLinearRelative.Done THEN
				pKuka.motion.KRC_MoveLinearRelative.ExecuteCmd := FALSE;
				cm.state := 1040;
			END_IF

		1040:
			cm.description := 'Close gripper and wait a little before moving to ensure proper grip';

			pKuka.gripperAction.action := CLOSE;

			pKuka.TON.PT := REAL_TO_TIME(200); // in ms
			pKuka.TON.IN := TRUE;
			IF pKuka.TON.Q THEN
				pKuka.TON.IN := FALSE;
				cm.state := 1050;
			END_IF

		1050:
			cm.description := 'Move to approach point of magazine with relative linear movement';

			// Almost everythings is already set from previous relative linear movement
			pKuka.tempPosition.Z := -45; // Move 100 mm backwards to magazine approach position
			// Status and turn is already set from moving to approach point

			pKuka.motion.KRC_MoveLinearRelative.Position := pKuka.tempPosition;

			pKuka.motion.KRC_MoveLinearRelative.ExecuteCmd := TRUE;
			IF pKuka.motion.KRC_MoveLinearRelative.Done THEN
				pKuka.motion.KRC_MoveLinearRelative.ExecuteCmd := FALSE;
				cm.state := 1060;
			END_IF

		1060:
			cm.description := 'Move to approach point of workstation with absolute linear movement';

			pKuka.convert.ValuesToCOORDSYS.Base := 1; // ACOPOS6D frame
			pKuka.convert.ValuesToCOORDSYS.IPO_Mode := 0; // #BASE
			pKuka.convert.ValuesToCOORDSYS();

			pKuka.convert.ValuesToPosition.posType := APPROACH_WORKSTATION;
			pKuka.convert.ValuesToPosition();

			pKuka.tempPosition := pKuka.convert.ValuesToPosition.outputPos;

			pKuka.motion.KRC_MoveLinearAbsolute.CoordinateSystem := pKuka.convert.ValuesToCOORDSYS.COORDSYS;
			pKuka.motion.KRC_MoveLinearAbsolute.Position := pKuka.tempPosition;

			pKuka.motion.KRC_MoveLinearAbsolute.ExecuteCmd := TRUE;
			IF pKuka.motion.KRC_MoveLinearAbsolute.Done THEN
				pKuka.motion.KRC_MoveLinearAbsolute.ExecuteCmd := FALSE;
				cm.state := 1070;
			END_IF

		1070:
			cm.description := 'Move to placement point at workstation with relative linear movement';

			pKuka.convert.ValuesToCOORDSYS.IPO_Mode := 1; // #TOOL
			pKuka.convert.ValuesToCOORDSYS();

			pKuka.motion.KRC_MoveLinearRelative.CoordinateSystem := pKuka.convert.ValuesToCOORDSYS.COORDSYS;

			pKuka.tempPosition.X := pKuka.tempPosition.Y := pKuka.tempPosition.Z := pKuka.tempPosition.A := pKuka.tempPosition.B := pKuka.tempPosition.C
				:= 0;
			pKuka.tempPosition.Z := 45; // Move 100 mm forwards to placement position
			// Status and turn is already set from moving to approach point

			pKuka.motion.KRC_MoveLinearRelative.Position := pKuka.tempPosition;

			pKuka.motion.KRC_MoveLinearRelative.ExecuteCmd := TRUE;
			IF pKuka.motion.KRC_MoveLinearRelative.Done THEN
				pKuka.motion.KRC_MoveLinearRelative.ExecuteCmd := FALSE;
				cm.state := 1080;
			END_IF

		1080:
			cm.description := 'Open gripper and wait a little before moving to ensure proper grip';

			pKuka.gripperAction.action := OPEN;

			pKuka.TON.PT := REAL_TO_TIME(200); // in ms
			pKuka.TON.IN := TRUE;
			IF pKuka.TON.Q THEN
				pKuka.TON.IN := FALSE;
				cm.state := 1090;
			END_IF

		1090:
			cm.description := 'Move to approach point of workkstation with relative linear movement';

			// Almost everythings is already set from previous relative linear movement
			pKuka.tempPosition.Z := -45; // Move 100 mm backwards to magazine approach position
			// Status and turn is already set from moving to approach point

			pKuka.motion.KRC_MoveLinearRelative.Position := pKuka.tempPosition;

			pKuka.motion.KRC_MoveLinearRelative.ExecuteCmd := TRUE;
			IF pKuka.motion.KRC_MoveLinearRelative.Done THEN
				pKuka.motion.KRC_MoveLinearRelative.ExecuteCmd := FALSE;
				robotOperating[i] := FALSE; // Set to false to allow shuttle to move away
				cm.state := 1100;
			END_IF

		1100:
			cm.description := 'Move to default point with absolute joint movement';

			pKuka.convert.ValuesToCOORDSYS.Base := 0; // World frame
			pKuka.convert.ValuesToCOORDSYS.IPO_Mode := 0; // #BASE
			pKuka.convert.ValuesToCOORDSYS();

			pKuka.convert.ValuesToPosition.posType := DEFAULT;
			pKuka.convert.ValuesToPosition();

			pKuka.tempPosition := pKuka.convert.ValuesToPosition.outputPos;

			pKuka.motion.KRC_MoveDirectAbsolute.CoordinateSystem := pKuka.convert.ValuesToCOORDSYS.COORDSYS;
			pKuka.motion.KRC_MoveDirectAbsolute.Position := pKuka.tempPosition;

			pKuka.motion.KRC_MoveDirectAbsolute.ExecuteCmd := TRUE;
			IF pKuka.motion.KRC_MoveDirectAbsolute.Done THEN
				pKuka.motion.KRC_MoveDirectAbsolute.ExecuteCmd := FALSE;
				cm.state := 1010;
			END_IF

	END_CASE

	pKuka.motion.KRC_MoveLinearAbsolute();
	pKuka.motion.KRC_MoveLinearRelative();
	pKuka.motion.KRC_MoveDirectAbsolute();
	pKuka.gripperAction();
	pKuka.TON();

END_ACTION
```

#### KUKADrilling.st - not listed in the package file held
```iecst
ACTION KUKADrilling:

	CASE cm.state OF

		1000:
			cm.description := 'Initialising parameters';

			pKuka.convert.ValuesToCOORDSYS.Tool := 1;
			pKuka.convert.ValuesToCOORDSYS();

			pKuka.convert.ValuesToPosition.axisGroupIdx := pKuka.axisGroupIdx;
			pKuka.convert.ValuesToPosition();

			pKuka.motion.KRC_MoveDirectAbsolute.AxisGroupIdx := pKuka.motion.KRC_MoveLinearAbsolute.AxisGroupIdx := pKuka.motion.KRC_MoveLinearRelative.AxisGroupIdx
				:=  pKuka.axisGroupIdx;
			pKuka.motion.KRC_MoveDirectAbsolute.KRC_AxisGroupRefArr := pKuka.motion.KRC_MoveLinearAbsolute.KRC_AxisGroupRefArr := pKuka.motion.KRC_MoveLinearRelative.KRC_AxisGroupRefArr
				:= ADR(AxisRef);
			pKuka.motion.KRC_MoveDirectAbsolute.Velocity := pKuka.motion.KRC_MoveLinearAbsolute.Velocity := pKuka.motion.KRC_MoveLinearRelative.Velocity
				:= 5; // Velocity in percent
			pKuka.motion.KRC_MoveDirectAbsolute.Acceleration := pKuka.motion.KRC_MoveLinearAbsolute.Acceleration := pKuka.motion.KRC_MoveLinearRelative.Acceleration
				:= 20; // Acceleration in percent
			pKuka.motion.KRC_MoveDirectAbsolute.BufferMode := pKuka.motion.KRC_MoveLinearAbsolute.BufferMode := pKuka.motion.KRC_MoveLinearRelative.BufferMode
				:= 2; // BUFFERED
			pKuka.motion.KRC_MoveLinearAbsolute.OriType := pKuka.motion.KRC_MoveLinearRelative.OriType
				:= 0; // 0: VAR | 1: CONSTANT | 2: JOINT
			pKuka.motion.KRC_MoveDirectAbsolute.ExecuteCmd := pKuka.motion.KRC_MoveLinearAbsolute.ExecuteCmd := pKuka.motion.KRC_MoveLinearRelative.ExecuteCmd
				:= FALSE;

			cm.state := 1010;

		1010:
			cm.description := 'Waiting for flag to start movement';

			IF robotOperating[i] THEN
				holeCounter := 0;
				cm.state := 1020;
			END_IF

		1020:
			cm.description := 'Move to first drilling approach point with absolute joint movement';

			pKuka.convert.ValuesToCOORDSYS.Base := 1; // ACOPOS6D frame
			pKuka.convert.ValuesToCOORDSYS.IPO_Mode := 0; // #BASE
			pKuka.convert.ValuesToCOORDSYS();

			pKuka.convert.ValuesToPosition.posType := APPROACH_WORKSTATION;
			pKuka.convert.ValuesToPosition();

			pKuka.tempPosition := pKuka.convert.ValuesToPosition.outputPos;

			pKuka.motion.KRC_MoveDirectAbsolute.CoordinateSystem := pKuka.convert.ValuesToCOORDSYS.COORDSYS;
			pKuka.motion.KRC_MoveDirectAbsolute.Position := pKuka.tempPosition;

			pKuka.motion.KRC_MoveDirectAbsolute.ExecuteCmd := TRUE;
			IF pKuka.motion.KRC_MoveDirectAbsolute.Done THEN
				pKuka.motion.KRC_MoveDirectAbsolute.ExecuteCmd := FALSE;
				cm.state := 1030;
			END_IF

		1030:
			cm.description := 'Move down to imitate drilling two holes using relative linear movement';

			pKuka.convert.ValuesToCOORDSYS.IPO_Mode := 1; // #TOOL
			pKuka.convert.ValuesToCOORDSYS();

			pKuka.motion.KRC_MoveLinearRelative.CoordinateSystem := pKuka.convert.ValuesToCOORDSYS.COORDSYS;

			pKuka.tempPosition.X := pKuka.tempPosition.Y := pKuka.tempPosition.Z := pKuka.tempPosition.A := pKuka.tempPosition.B := pKuka.tempPosition.C
				:= 0;
			pKuka.tempPosition.Z := 100; // Move 100 mm forwards to pickup position
			// Status and turn is already set from moving to approach point

			pKuka.motion.KRC_MoveLinearRelative.Position := pKuka.tempPosition;

			pKuka.motion.KRC_MoveLinearRelative.ExecuteCmd := TRUE;
			IF pKuka.motion.KRC_MoveLinearRelative.Done THEN
				pKuka.motion.KRC_MoveLinearRelative.ExecuteCmd := FALSE;
				cm.state := 1040;
			END_IF

		1040:
			cm.description := 'Move back up again with relative linear movement';

			// Almost everythings is already set from previous relative linear movement
			pKuka.tempPosition.Z := -100; // Move 100 mm backwards to magazine approach position
			// Status and turn is already set from moving to approach point

			pKuka.motion.KRC_MoveLinearRelative.Position := pKuka.tempPosition;

			pKuka.motion.KRC_MoveLinearRelative.ExecuteCmd := TRUE;
			IF pKuka.motion.KRC_MoveLinearRelative.Done THEN
				pKuka.motion.KRC_MoveLinearRelative.ExecuteCmd := FALSE;

				holeCounter := holeCounter + 2;

				IF holeCounter = orderSpec[i] THEN
					cm.state := 1060;
				ELSE
					cm.state := 1050;
				END_IF

			END_IF

		1050:
			cm.description := 'Move to second drilling approach point with relative linear movement';

			pKuka.tempPosition.X := pKuka.tempPosition.Y := pKuka.tempPosition.Z := pKuka.tempPosition.A := pKuka.tempPosition.B := pKuka.tempPosition.C
				:= 0;
			pKuka.tempPosition.Y := 100; // Move 100 mm laterally to pickup position (NEED TO CHANGE)
			// Status and turn is already set from moving to approach point

			pKuka.motion.KRC_MoveLinearRelative.Position := pKuka.tempPosition;

			pKuka.motion.KRC_MoveLinearRelative.ExecuteCmd := TRUE;
			IF pKuka.motion.KRC_MoveLinearRelative.Done THEN
				pKuka.motion.KRC_MoveLinearRelative.ExecuteCmd := FALSE;
				cm.state := 1030;
			END_IF

		1060:
			cm.description := 'Move to default point with absolute joint movement';

			pKuka.convert.ValuesToCOORDSYS.Base := 0; // World frame
			pKuka.convert.ValuesToCOORDSYS.IPO_Mode := 0; // #BASE
			pKuka.convert.ValuesToCOORDSYS();

			pKuka.convert.ValuesToPosition.posType := DEFAULT;
			pKuka.convert.ValuesToPosition();

			pKuka.tempPosition := pKuka.convert.ValuesToPosition.outputPos;

			pKuka.motion.KRC_MoveDirectAbsolute.CoordinateSystem := pKuka.convert.ValuesToCOORDSYS.COORDSYS;
			pKuka.motion.KRC_MoveDirectAbsolute.Position := pKuka.tempPosition;

			pKuka.motion.KRC_MoveDirectAbsolute.ExecuteCmd := TRUE;
			IF pKuka.motion.KRC_MoveDirectAbsolute.Done THEN
				pKuka.motion.KRC_MoveDirectAbsolute.ExecuteCmd := FALSE;
				pKuka.cm.state := 1010;
			END_IF

	END_CASE

	pKuka.motion.KRC_MoveLinearAbsolute();
	pKuka.motion.KRC_MoveLinearRelative();
	pKuka.motion.KRC_MoveDirectAbsolute();

END_ACTION
```

#### KUKAFuse.st - not listed in the package file held
```iecst
ACTION KUKAFuse:

END_ACTION
```

#### KUKAPcb.st - not listed in the package file held
```iecst
ACTION KUKAPcb:

	CASE cm.state OF

		1000:
			cm.description := 'Initialising parameters';

			pKuka.convert.ValuesToCOORDSYS.Tool := 1;
			pKuka.convert.ValuesToCOORDSYS();

			pKuka.convert.ValuesToPosition.axisGroupIdx := pKuka.axisGroupIdx;
			pKuka.convert.ValuesToPosition();

			pKuka.motion.KRC_MoveDirectAbsolute.AxisGroupIdx := pKuka.motion.KRC_MoveLinearAbsolute.AxisGroupIdx := pKuka.motion.KRC_MoveLinearRelative.AxisGroupIdx
				:=  pKuka.axisGroupIdx;
			pKuka.motion.KRC_MoveDirectAbsolute.KRC_AxisGroupRefArr := pKuka.motion.KRC_MoveLinearAbsolute.KRC_AxisGroupRefArr := pKuka.motion.KRC_MoveLinearRelative.KRC_AxisGroupRefArr
				:= ADR(AxisRef);
			pKuka.motion.KRC_MoveDirectAbsolute.Velocity := pKuka.motion.KRC_MoveLinearAbsolute.Velocity := pKuka.motion.KRC_MoveLinearRelative.Velocity
			:= 10; // Velocity in percent
			pKuka.motion.KRC_MoveDirectAbsolute.Acceleration := pKuka.motion.KRC_MoveLinearAbsolute.Acceleration := pKuka.motion.KRC_MoveLinearRelative.Acceleration
				:= 20; // Acceleration in percent
			pKuka.motion.KRC_MoveDirectAbsolute.BufferMode := pKuka.motion.KRC_MoveLinearAbsolute.BufferMode := pKuka.motion.KRC_MoveLinearRelative.BufferMode
				:= 2; // BUFFERED
			pKuka.motion.KRC_MoveLinearAbsolute.OriType := pKuka.motion.KRC_MoveLinearRelative.OriType
				:= 0; // 0: VAR | 1: CONSTANT | 2: JOINT
			pKuka.motion.KRC_MoveDirectAbsolute.ExecuteCmd := pKuka.motion.KRC_MoveLinearAbsolute.ExecuteCmd := pKuka.motion.KRC_MoveLinearRelative.ExecuteCmd
				:= FALSE;

			cm.state := 1010;

		1010:
			cm.description := 'Waiting for flag to start movement';

			IF robotOperating[i] THEN
				cm.state := 1020;
			END_IF

		1020:
			cm.description := 'Move to approach point of magazine with absolute joint movement';

			pKuka.convert.ValuesToCOORDSYS.Base := 2; // Magazine frame
			pKuka.convert.ValuesToCOORDSYS.IPO_Mode := 0; // #BASE
			pKuka.convert.ValuesToCOORDSYS();

			pKuka.convert.ValuesToPosition.posType := APPROACH_MAGAZINE;
			pKuka.convert.ValuesToPosition();

			pKuka.tempPosition := pKuka.convert.ValuesToPosition.outputPos;

			pKuka.motion.KRC_MoveDirectAbsolute.CoordinateSystem := pKuka.convert.ValuesToCOORDSYS.COORDSYS;
			pKuka.motion.KRC_MoveDirectAbsolute.Position := pKuka.tempPosition;

			pKuka.motion.KRC_MoveDirectAbsolute.ExecuteCmd := TRUE;
			IF pKuka.motion.KRC_MoveDirectAbsolute.Done THEN
				pKuka.motion.KRC_MoveDirectAbsolute.ExecuteCmd := FALSE;
				cm.state := 1030;
			END_IF

		1030:
			cm.description := 'Move to pickup point at magazine with relative linear movement';

			pKuka.convert.ValuesToCOORDSYS.IPO_Mode := 1; // #TOOL
			pKuka.convert.ValuesToCOORDSYS();

			pKuka.motion.KRC_MoveLinearRelative.CoordinateSystem := pKuka.convert.ValuesToCOORDSYS.COORDSYS;

			pKuka.tempPosition.X := pKuka.tempPosition.Y := pKuka.tempPosition.Z := pKuka.tempPosition.A := pKuka.tempPosition.B := pKuka.tempPosition.C
				:= 0;
			pKuka.tempPosition.Z := -relativeDistance; // Move 100 mm forwards to pickup position
			// Status and turn is already set from moving to approach point

			pKuka.motion.KRC_MoveLinearRelative.Position := pKuka.tempPosition;

			pKuka.motion.KRC_MoveLinearRelative.ExecuteCmd := TRUE;
			IF pKuka.motion.KRC_MoveLinearRelative.Done THEN
				pKuka.motion.KRC_MoveLinearRelative.ExecuteCmd := FALSE;
				cm.state := 1040;
			END_IF

		1040:
			cm.description := 'Close gripper and wait a little before moving to ensure proper grip';

			pKuka.gripperAction.action := CLOSE;

			pKuka.TON.PT := REAL_TO_TIME(200); // in ms
			pKuka.TON.IN := TRUE;
			IF pKuka.TON.Q THEN
				pKuka.TON.IN := FALSE;
				cm.state := 1050;
			END_IF

		1050:
			cm.description := 'Move to approach point of magazine with relative linear movement';

			// Almost everythings is already set from previous relative linear movement
			pKuka.tempPosition.Z := relativeDistance; // Move 100 mm backwards to magazine approach position
			// Status and turn is already set from moving to approach point

			pKuka.motion.KRC_MoveLinearRelative.Position := pKuka.tempPosition;

			pKuka.motion.KRC_MoveLinearRelative.ExecuteCmd := TRUE;
			IF pKuka.motion.KRC_MoveLinearRelative.Done THEN
				pKuka.motion.KRC_MoveLinearRelative.ExecuteCmd := FALSE;
				cm.state := 1060;
			END_IF

		1060:
			cm.description := 'Move to approach point of workstation with absolute linear movement';

			pKuka.convert.ValuesToCOORDSYS.Base := 1; // ACOPOS6D frame
			pKuka.convert.ValuesToCOORDSYS.IPO_Mode := 0; // #BASE
			pKuka.convert.ValuesToCOORDSYS();

			pKuka.convert.ValuesToPosition.posType := APPROACH_WORKSTATION;
			pKuka.convert.ValuesToPosition();

			pKuka.tempPosition := pKuka.convert.ValuesToPosition.outputPos;

			pKuka.motion.KRC_MoveLinearAbsolute.CoordinateSystem := pKuka.convert.ValuesToCOORDSYS.COORDSYS;
			pKuka.motion.KRC_MoveLinearAbsolute.Position := pKuka.tempPosition;

			pKuka.motion.KRC_MoveLinearAbsolute.ExecuteCmd := TRUE;
			IF pKuka.motion.KRC_MoveLinearAbsolute.Done THEN
				pKuka.motion.KRC_MoveLinearAbsolute.ExecuteCmd := FALSE;
				cm.state := 1070;
			END_IF

		1070:
			cm.description := 'Move to placement point at workstation with relative linear movement';

			pKuka.convert.ValuesToCOORDSYS.IPO_Mode := 1; // #TOOL
			pKuka.convert.ValuesToCOORDSYS();

			pKuka.motion.KRC_MoveLinearRelative.CoordinateSystem := pKuka.convert.ValuesToCOORDSYS.COORDSYS;

			pKuka.tempPosition.X := pKuka.tempPosition.Y := pKuka.tempPosition.Z := pKuka.tempPosition.A := pKuka.tempPosition.B := pKuka.tempPosition.C
				:= 0;
			pKuka.tempPosition.Z := -relativeDistance; // Move 80 mm forwards to placement position
			// Status and turn is already set from moving to approach point

			pKuka.motion.KRC_MoveLinearRelative.Position := pKuka.tempPosition;

			pKuka.motion.KRC_MoveLinearRelative.ExecuteCmd := TRUE;
			IF pKuka.motion.KRC_MoveLinearRelative.Done THEN
				pKuka.motion.KRC_MoveLinearRelative.ExecuteCmd := FALSE;
				cm.state := 1080;
			END_IF

		1080:
			cm.description := 'Open gripper and wait a little before moving to ensure proper grip';

			pKuka.gripperAction.action := OPEN;

			pKuka.TON.PT := REAL_TO_TIME(200); // in ms
			pKuka.TON.IN := TRUE;
			IF pKuka.TON.Q THEN
				pKuka.TON.IN := FALSE;
				cm.state := 1090;
			END_IF

		1090:
			cm.description := 'Move to approach point of workkstation with relative linear movement';

			// Almost everythings is already set from previous relative linear movement
			pKuka.tempPosition.Z := relativeDistance; // Move 100 mm backwards to magazine approach position
			// Status and turn is already set from moving to approach point

			pKuka.motion.KRC_MoveLinearRelative.Position := pKuka.tempPosition;

			pKuka.motion.KRC_MoveLinearRelative.ExecuteCmd := TRUE;
			IF pKuka.motion.KRC_MoveLinearRelative.Done THEN
				pKuka.motion.KRC_MoveLinearRelative.ExecuteCmd := FALSE;
				robotOperating[i] := FALSE; // Set to false to allow shuttle to move away
				cm.state := 1100;
			END_IF

		1100:
			cm.description := 'Move to default point with absolute joint movement';

			pKuka.convert.ValuesToCOORDSYS.Base := 0; // World frame
			pKuka.convert.ValuesToCOORDSYS.IPO_Mode := 0; // #BASE
			pKuka.convert.ValuesToCOORDSYS();

			pKuka.convert.ValuesToPosition.posType := DEFAULT;
			pKuka.convert.ValuesToPosition();

			pKuka.tempPosition := pKuka.convert.ValuesToPosition.outputPos;

			pKuka.motion.KRC_MoveDirectAbsolute.CoordinateSystem := pKuka.convert.ValuesToCOORDSYS.COORDSYS;
			pKuka.motion.KRC_MoveDirectAbsolute.Position := pKuka.tempPosition;

			pKuka.motion.KRC_MoveDirectAbsolute.ExecuteCmd := TRUE;
			IF pKuka.motion.KRC_MoveDirectAbsolute.Done THEN
				pKuka.motion.KRC_MoveDirectAbsolute.ExecuteCmd := FALSE;
				cm.state := 1010;
			END_IF

	END_CASE

	pKuka.motion.KRC_MoveLinearAbsolute();
	pKuka.motion.KRC_MoveLinearRelative();
	pKuka.motion.KRC_MoveDirectAbsolute();
	pKuka.gripperAction();
	pKuka.TON();

END_ACTION
```

#### KUKATopCover.st - not listed in the package file held
```iecst
ACTION KUKATopCover:

END_ACTION
```

#### KUKAUnloading.st - not listed in the package file held
```iecst
ACTION KUKAUnloading:

END_ACTION
```

#### mxA_ErrorMessage.st - not listed in the package file held
```iecst
ACTION mxA_ErrorMessage:

	CASE step_UDPConnect OF

		//////////////////////////////////////////////////////////
		//			Opening the 2 Ports to communicate			//
		//	Port 55555 is used for Receiving					//
		//	Port 50055 is used for Sending						//
		//////////////////////////////////////////////////////////
		STATE_OPEN:
			UdpOpen_0.enable := 1; 										//opening port for Receiving
			UdpOpen_0.port := 55555;
			UdpOpen_0();

			UdpOpen_1.enable := 1;  									//opening port for Sending
			UdpOpen_1.port := 50055;
			UdpOpen_1();

			IF UdpOpen_0.status = ERR_OK AND UdpOpen_1.status = ERR_OK THEN		//if both ports are open send request
				step_UDPConnect := STATE_WAIT;
			END_IF

		//////////////////////////////////////////////////////////
		//		Waiting State for the manual trigger			//
		//		to get all the Messages	 (request)				//
		//////////////////////////////////////////////////////////
		STATE_WAIT:

			TON_0.IN := 0;

			IF ReloadMsg = 1 OR WorkAroundCounter = 1 THEN				//Var WorkAroundCounter is just a Workaround to Reload the messages 2 times
				step_UDPConnect := STATE_SEND;							// otherwise messages are displayed when requensting the first time!
			END_IF

			IF WorkAroundCounter >= 2 THEN
				WorkAroundCounter := 0;
			END_IF

		//////////////////////////////////////////////////////////
		//		Sending the Message to the KRC to 				//
		//		get all the Messages							//
		//////////////////////////////////////////////////////////
		STATE_SEND:

			FOR counterMsg := 0 TO 15 DO						//Reseting the Array with the Messages
				TextArray[counterMsg] := '';
			END_FOR

			i := 0;												//Reseting counter for the Message Array
			MsgToKrc := 'GetAllKrcMessages';					//Message to KRC -> to get the Messages from KRC

			UdpSend_0.enable := 1;
			UdpSend_0.ident := UdpOpen_1.ident;
			UdpSend_0.pHost := ADR('192.168.1.2');
			UdpSend_0.port := 50055;
			UdpSend_0.pData := ADR(MsgToKrc);
			UdpSend_0.datalen := SIZEOF(MsgToKrc);
			UdpSend_0();

			IF UdpSend_0.status = ERR_OK THEN					//ERR_OK -> NO ERROR
				WorkAroundCounter := WorkAroundCounter +1;
				step_UDPConnect := STATE_RECEIVE;
			END_IF

		//////////////////////////////////////////////////////////
		//		Receiving the Messages from KRC					//
		//		Per cycle 1 msg will be received				//
		// 		If no message after 1s change to STATE_WAIT		//
		//////////////////////////////////////////////////////////
		STATE_RECEIVE:
			UdpRecv_0.enable := 1;
			UdpRecv_0.ident := UdpOpen_0.ident;
			UdpRecv_0.pData := ADR(InputUDPString);
			UdpRecv_0.datamax := 255;
			UdpRecv_0();

			IF UdpRecv_0.status = ERR_OK THEN					//ERR_OK -> NO ERROR

				InputUDPString 	:= LEFT(InputUDPString, UDINT_TO_INT(UdpRecv_0.recvlen));
				TON_0.IN 		:= 0; // Reset timer - msg received
				step_UDPConnect 		:= STATE_DISPLAY;

			ELSIF (UdpRecv_0.status = udpERR_NO_DATA) THEN

				TON_0.IN := 1; // set timer - no msg available, after 1 sec change state to wait
				TON_0.PT := T#1s;

			END_IF

			// check if timer is set to true
			IF TON_0.Q = 1 THEN

				step_UDPConnect := STATE_WAIT;
			END_IF

		//////////////////////////////////////////////////////////
		//		State to transfer the Message					//
		//		to the Array which is displayed at Visu			//
		//////////////////////////////////////////////////////////
		STATE_DISPLAY:

			TextArray[i] := InputUDPString;								//write current message to array to display
			IF i >= 14 THEN
				i := 0;
			ELSE
				memset(ADR(InputUDPString),0,SIZEOF(InputUDPString));	//Clear / Reset the input of the Variable
				i := i + 1;
				step_UDPConnect := STATE_RECEIVE;						//Go to Receive state, to see if another message available
			END_IF;

	END_CASE;

	//Call of the Timer for the TimeOut when no Message
	TON_0();

END_ACTION
```

#### mxA_JointMovement.st - not listed in the package file held
```iecst
ACTION mxA_JointMovement:

	CASE KUKAs[i].cm.state OF

		0:
			// Waiting for robot 1 to be ready to move
			IF 	KUKAs[i].status.P_ AND KUKAs[i].status.S_ AND KUKAs[i].status.R_ AND KUKAs[i].status.I_ AND KUKAs[i].status.EXT_ THEN
				KUKAs[i].cm.state := 10;
			END_IF

		10:
			// Set initial parameters for movement
			KUKAs[i].motion.KRC_MoveAxisAbsolute.ExecuteCmd 			:= FALSE;
			KUKAs[i].motion.KRC_MoveAxisAbsolute.AxisGroupIdx 			:= KUKAs[i].AxisGroupIdx;
			KUKAs[i].motion.KRC_MoveAxisAbsolute.KRC_AxisGroupRefArr	:= ADR(AxisRef);
			KUKAs[i].motion.KRC_MoveAxisAbsolute.Velocity 				:= 10;
			KUKAs[i].motion.KRC_MoveAxisAbsolute.Acceleration 			:= 20;
			KUKAs[i].motion.KRC_MoveAxisAbsolute.BufferMode 			:= 2;

			position1.A1 := 0;
			position1.A2 := -70;
			position1.A3 := 90;
			position1.A4 := 0;
			position1.A5 := -90;
			position1.A6 := 0;

			position2.A1 := 0;
			position2.A2 := -90;
			position2.A3 := 90;
			position2.A4 := 0;
			position2.A5 := 80;
			position2.A6 := 0;

			KUKAs[i].cm.state := 20;

		20: // Set initial position
			KUKAs[i].motion.KRC_MoveAxisAbsolute.AxisPosition := position1;

			KUKAs[i].motion.KRC_MoveAxisAbsolute.ExecuteCmd 	:= TRUE;
			IF KUKAs[i].motion.KRC_MoveAxisAbsolute.Done THEN
				KUKAs[i].motion.KRC_MoveAxisAbsolute.ExecuteCmd := FALSE;
				KUKAs[i].cm.state := 30;
			END_IF

		30:	// Set second position
			KUKAs[i].motion.KRC_MoveAxisAbsolute.AxisPosition := position2;

			KUKAs[i].motion.KRC_MoveAxisAbsolute.ExecuteCmd	:= TRUE;
			IF KUKAs[i].motion.KRC_MoveAxisAbsolute.Done THEN
				KUKAs[i].motion.KRC_MoveAxisAbsolute.ExecuteCmd	:= FALSE;
				KUKAs[i].cm.state := 20;
			END_IF

	END_CASE

	mxa_ValuesToCOORDSYS_0();
	KUKAs[i].motion.KRC_MoveAxisAbsolute();

END_ACTION
```

#### mxA_KUKA1.st - not listed in the package file held
```iecst
ACTION mxA_KUKA1:

	CASE cm.state OF
		0: // Wait for the robot to be ready
			IF 	pKuka.status.P_ AND pKuka.status.S_ AND pKuka.status.R_ AND pKuka.status.I_ AND pKuka.status.EXT_ THEN
				pKuka.cm.state := 10;
			END_IF

		10: // Wait for "perform proccess" flag from shuttle

		20: // Perform movement 1

		30: // Perform movement 2

		40: // Perform movement n and set "process done" flag, allowing the shuttle to move

		50: // Move to appropriate start position (e.g. near fixtures) and set "workstation ready" flag
			cm.state := 10;

	END_CASE

END_ACTION
```

#### mxA_KUKA2.st - not listed in the package file held
```iecst
ACTION mxA_KUKA2:

END_ACTION
```

#### mxA_KUKA3.st - not listed in the package file held
```iecst
ACTION mxA_KUKA3:

END_ACTION
```

#### mxA_KUKA4.st - not listed in the package file held
```iecst
ACTION mxA_KUKA4:

END_ACTION
```

#### mxA_KUKA5.st - not listed in the package file held
```iecst
ACTION mxA_KUKA5:

END_ACTION
```

#### mxA_KUKA6.st - not listed in the package file held
```iecst
ACTION mxA_KUKA6:

END_ACTION
```

#### mxA_LinearMovement.st - not listed in the package file held
```iecst
ACTION mxA_LinearMovement:

	CASE KUKAs[i].cm.state OF

		0:
			// Waiting for robot 1 to be ready to move
			IF 	KUKAs[i].status.P_ AND KUKAs[i].status.S_ AND KUKAs[i].status.I_ AND KUKAs[i].status.R_ AND KUKAs[i].status.EXT_ THEN
				KUKAs[i].cm.state := 10;
			END_IF

		10:
			toolCover.X := 0;
			toolCover.Y := 0;
			toolCover.Z := 100;
			toolCover.A := 0;
			toolCover.B := 0;
			toolCover.C := 0;

			KRC_Write_Tool_Data.AxisGroupIdx 		:= KUKAs[i].AxisGroupIdx;
			KRC_Write_Tool_Data.KRC_AxisGroupRefArr := ADR(AxisRef);
			KRC_Write_Tool_Data.ToolNo 				:= 1;
			KRC_Write_Tool_Data.ToolData 			:= toolCover;
			KRC_Write_Tool_Data.BufferMode 			:= 2;
			KRC_Write_Tool_Data.ExecuteCmd			:= TRUE;

			IF KRC_Write_Tool_Data.Done THEN
				KRC_Write_Tool_Data.ExecuteCmd		:= FALSE;
				KUKAs[i].cm.state := 20;
			END_IF

		20:

			//Set frames as coordsys
			mxa_ValuesToCOORDSYS_0.Tool 	:= 1; // Change to 1 when it works
			mxa_ValuesToCOORDSYS_0.Base 	:= 1;
			mxa_ValuesToCOORDSYS_0.IPO_Mode := 0;

			KUKAs[i].cm.state := 30;

		30:

			coordSys := mxa_ValuesToCOORDSYS_0.COORDSYS;

			KUKAs[i].motion.KRC_MoveLinearAbsolute.AxisGroupIdx 		:= KUKAs[i].AxisGroupIdx;
			KUKAs[i].motion.KRC_MoveLinearAbsolute.KRC_AxisGroupRefArr	:= ADR(AxisRef);
			KUKAs[i].motion.KRC_MoveLinearAbsolute.Velocity				:= 10;
			KUKAs[i].motion.KRC_MoveLinearAbsolute.Acceleration  		:= 20;
			KUKAs[i].motion.KRC_MoveLinearAbsolute.CoordinateSystem		:= coordSys;
			KUKAs[i].motion.KRC_MoveLinearAbsolute.OriType 				:= 0;
			KUKAs[i].motion.KRC_MoveLinearAbsolute.BufferMode			:= 2;

			KUKAs[i].cm.state := 40;

		40:
			endPOS.X := 302;
			endPOS.Y := -2;
			endPOS.Z := 527;
			endPOS.A := -178;
			endPOS.B := 26;
			endPOS.C := -178;
			endPOS.Status := 2; //010
			endPOS.Turn := 2; //000010

			KUKAs[i].motion.KRC_MoveLinearAbsolute.Position			:= endPOS;

			KUKAs[i].motion.KRC_MoveLinearAbsolute.ExecuteCmd 		:= TRUE;
			IF KUKAs[i].motion.KRC_MoveLinearAbsolute.Done THEN
				KUKAs[i].motion.KRC_MoveLinearAbsolute.ExecuteCmd 	:= FALSE;
				KUKAs[i].cm.state := 50;
			END_IF

		50:
			endPOS.X := 430;
			endPOS.Y := -2;
			endPOS.Z := 527;
			endPOS.A := -178;
			endPOS.B := 26;
			endPOS.C := -178;
			endPOS.Status := 2; //010
			endPOS.Turn := 2; //000010

			KUKAs[i].motion.KRC_MoveLinearAbsolute.Position			:= endPOS;

			KUKAs[i].motion.KRC_MoveLinearAbsolute.ExecuteCmd 		:= TRUE;
			IF KUKAs[i].motion.KRC_MoveLinearAbsolute.Done THEN
				KUKAs[i].motion.KRC_MoveLinearAbsolute.ExecuteCmd 	:= FALSE;
				KUKAs[i].cm.state 	:= 40;
			END_IF

	END_CASE

	KRC_Write_Tool_Data();
	mxa_ValuesToCOORDSYS_0();
	KUKAs[i].motion.KRC_MoveLinearAbsolute();

END_ACTION
```
